Universal Robots URScript: azat-test-new.script

def azattestnew():
  set_gravity([0.0, 0.0, 9.82])
  set_safety_mode_transition_hardness(1)
  set_target_payload(1.070000, [0.002000, 0.003000, 0.057000], [0.001723, 0.001723, 0.001723, 0.000000, 0.000000, 0.000000])
  step_count_12e684db_e6cc_44c8_bfb7_09d4b2be2b77 = 0.0
  thread Step_Counter_Thread_decf62d9_1c1e_413a_991a_3884a730e61c():
    while (True):
      step_count_12e684db_e6cc_44c8_bfb7_09d4b2be2b77 = step_count_12e684db_e6cc_44c8_bfb7_09d4b2be2b77 + 1.0
      sync()
    end
  end
  run Step_Counter_Thread_decf62d9_1c1e_413a_991a_3884a730e61c()
  set_tool_communication(True, 1000000, 2, 1, 1.5, 3.5)
  set_tool_output_mode(0)
  set_tool_digital_output_mode(0, 1)
  set_tool_digital_output_mode(1, 1)
  set_tool_voltage(0)
  set_standard_analog_input_domain(0, 1)
  set_standard_analog_input_domain(1, 1)
  set_tool_analog_input_domain(0, 1)
  set_tool_analog_input_domain(1, 1)
  set_analog_outputdomain(0, 0)
  set_analog_outputdomain(1, 0)
  set_input_actions_to_default()
  set_tcp(p[0.0,0.0,0.0,0.0,0.0,0.0])
  global Plane_1=p[-0.700006141123905,1.3454883874109249E-6,0.3910559577028425,-1.2089868272251132,-1.2089999932245832,1.20858562628424]
  global Plane_2=p[0.0,0.0,0.0,0.0,0.0,0.0]
  global Point_1=p[0.6913645118948067,-0.12399382748223003,0.49223711947071,-1.2983729986843258,1.1259514972191385,-1.2203503861141718]
  $ 1 "Robot Program"
  $ 2 "Script: bookmark_jonathan.script"
  def Machining1():
    # Default parameters:
    global speed_ms = 0.3
    global speed_rads = 0.75
    global accel_mss = 3
    global accel_radss = 1.2
    global blend_radius_m = 0.001

    # Add subprograms here
    # Start of main program
    # Program generated by RoboDK v5.6.5 for UR10e on 13/10/2023 15:41:24
    # Using nominal kinematics.
    blend_radius_m = 0.001
    speed_ms = 1.000
    # set_reference(p[0.335000, -0.154000, 0.001500, 0.000000, 0.000000, 0.000000])
    set_tcp(p[0.000000, 0.000000, 0.252000, 0.000000, 0.000000, 0.000000])
    # Show Tool
    movej([0.110042, -1.089243, -2.581851, -1.041295, 1.570796, 1.680839],accel_radss,speed_rads,0,blend_radius_m)
    movel([0.110042, -1.182009, -2.646989, -0.883391, 1.570796, 1.680839],accel_mss,speed_ms,0,blend_radius_m)
    speed_ms = 1.000
    movel([0.110042, -1.209222, -2.661511, -0.841656, 1.570796, 1.680839],accel_mss,speed_ms,0,blend_radius_m)
    speed_ms = 0.003
    movel([0.110042, -1.219969, -2.666830, -0.825590, 1.570796, 1.680839],accel_mss,speed_ms,0,blend_radius_m)
    speed_ms = 0.007
    movel([0.109778, -1.220368, -2.666631, -0.825390, 1.570796, 1.680574],accel_mss,speed_ms,0,blend_radius_m)
    movel([0.108896, -1.220713, -2.666459, -0.825217, 1.570796, 1.679693],accel_mss,speed_ms,0,blend_radius_m)
    movel([0.108041, -1.221013, -2.666309, -0.825067, 1.570796, 1.678837],accel_mss,speed_ms,0,blend_radius_m)
    movel([0.107066, -1.221345, -2.666143, -0.824901, 1.570796, 1.677863],accel_mss,speed_ms,0,blend_radius_m)
    movel([0.105797, -1.221762, -2.665934, -0.824693, 1.570796, 1.676593],accel_mss,speed_ms,0,blend_radius_m)
    movel([0.105050, -1.221982, -2.665824, -0.824583, 1.570796, 1.675846],accel_mss,speed_ms,0,blend_radius_m)
    movel([0.104582, -1.222084, -2.665773, -0.824532, 1.570796, 1.675378],accel_mss,speed_ms,0,blend_radius_m)
    movel([0.104339, -1.221931, -2.665850, -0.824608, 1.570796, 1.675136],accel_mss,speed_ms,0,blend_radius_m)
    movel([0.104313, -1.221582, -2.666024, -0.824782, 1.570796, 1.675109],accel_mss,speed_ms,0,blend_radius_m)
    movel([0.104310, -1.221133, -2.666249, -0.825007, 1.570796, 1.675106],accel_mss,speed_ms,0,blend_radius_m)
    movel([0.104335, -1.220607, -2.666512, -0.825270, 1.570796, 1.675132],accel_mss,speed_ms,0,blend_radius_m)
    movel([0.104393, -1.219927, -2.666851, -0.825611, 1.570796, 1.675190],accel_mss,speed_ms,0,blend_radius_m)
    movel([0.104458, -1.219512, -2.667058, -0.825819, 1.570796, 1.675255],accel_mss,speed_ms,0,blend_radius_m)
    movel([0.104671, -1.219046, -2.667290, -0.826053, 1.570796, 1.675468],accel_mss,speed_ms,0,blend_radius_m)
    movel([0.104983, -1.218876, -2.667375, -0.826139, 1.570796, 1.675780],accel_mss,speed_ms,0,blend_radius_m)
    movel([0.105336, -1.218982, -2.667322, -0.826085, 1.570796, 1.676132],accel_mss,speed_ms,0,blend_radius_m)
    movel([0.105719, -1.218905, -2.667360, -0.826124, 1.570796, 1.676515],accel_mss,speed_ms,0,blend_radius_m)
    movel([0.106129, -1.218813, -2.667406, -0.826170, 1.570796, 1.676925],accel_mss,speed_ms,0,blend_radius_m)
    movel([0.106457, -1.218831, -2.667397, -0.826161, 1.570796, 1.677253],accel_mss,speed_ms,0,blend_radius_m)
    movel([0.106802, -1.218829, -2.667398, -0.826162, 1.570796, 1.677598],accel_mss,speed_ms,0,blend_radius_m)
    movel([0.107299, -1.218637, -2.667493, -0.826259, 1.570796, 1.678095],accel_mss,speed_ms,0,blend_radius_m)
    movel([0.107817, -1.218437, -2.667593, -0.826359, 1.570796, 1.678614],accel_mss,speed_ms,0,blend_radius_m)
    movel([0.108199, -1.218441, -2.667591, -0.826357, 1.570796, 1.678995],accel_mss,speed_ms,0,blend_radius_m)
    movel([0.108539, -1.218479, -2.667572, -0.826338, 1.570796, 1.679335],accel_mss,speed_ms,0,blend_radius_m)
    movel([0.108879, -1.218392, -2.667615, -0.826382, 1.570796, 1.679675],accel_mss,speed_ms,0,blend_radius_m)
    movel([0.109256, -1.218165, -2.667728, -0.826496, 1.570796, 1.680053],accel_mss,speed_ms,0,blend_radius_m)
    movel([0.109705, -1.217777, -2.667921, -0.826692, 1.570796, 1.680502],accel_mss,speed_ms,0,blend_radius_m)
    movel([0.110106, -1.217433, -2.668091, -0.826865, 1.570796, 1.680902],accel_mss,speed_ms,0,blend_radius_m)
    movel([0.110486, -1.217183, -2.668215, -0.826991, 1.570796, 1.681283],accel_mss,speed_ms,0,blend_radius_m)
    movel([0.110803, -1.217055, -2.668278, -0.827056, 1.570796, 1.681599],accel_mss,speed_ms,0,blend_radius_m)
    movel([0.111053, -1.217213, -2.668200, -0.826976, 1.570796, 1.681849],accel_mss,speed_ms,0,blend_radius_m)
    movel([0.110944, -1.217659, -2.667979, -0.826751, 1.570796, 1.681740],accel_mss,speed_ms,0,blend_radius_m)
    movel([0.110733, -1.218302, -2.667660, -0.826427, 1.570796, 1.681529],accel_mss,speed_ms,0,blend_radius_m)
    movel([0.110389, -1.219201, -2.667213, -0.825975, 1.570796, 1.681186],accel_mss,speed_ms,0,blend_radius_m)
    movel([0.110219, -1.219606, -2.667011, -0.825772, 1.570796, 1.681015],accel_mss,speed_ms,0,blend_radius_m)
    movel([0.110042, -1.219969, -2.666830, -0.825590, 1.570796, 1.680839],accel_mss,speed_ms,0,blend_radius_m)
    speed_ms = 0.003
    movel([0.110042, -1.223618, -2.668588, -0.820184, 1.570796, 1.680839],accel_mss,speed_ms,0,blend_radius_m)
    speed_ms = 0.007
    movel([0.109778, -1.224016, -2.668388, -0.819985, 1.570796, 1.680574],accel_mss,speed_ms,0,blend_radius_m)
    movel([0.108896, -1.224361, -2.668215, -0.819813, 1.570796, 1.679693],accel_mss,speed_ms,0,blend_radius_m)
    movel([0.108041, -1.224660, -2.668065, -0.819664, 1.570796, 1.678837],accel_mss,speed_ms,0,blend_radius_m)
    movel([0.107066, -1.224992, -2.667898, -0.819499, 1.570796, 1.677863],accel_mss,speed_ms,0,blend_radius_m)
    movel([0.105797, -1.225409, -2.667688, -0.819292, 1.570796, 1.676593],accel_mss,speed_ms,0,blend_radius_m)
    movel([0.105050, -1.225628, -2.667578, -0.819183, 1.570796, 1.675846],accel_mss,speed_ms,0,blend_radius_m)
    movel([0.104582, -1.225730, -2.667526, -0.819132, 1.570796, 1.675378],accel_mss,speed_ms,0,blend_radius_m)
    movel([0.104339, -1.225577, -2.667604, -0.819209, 1.570796, 1.675136],accel_mss,speed_ms,0,blend_radius_m)
    movel([0.104313, -1.225229, -2.667779, -0.819381, 1.570796, 1.675109],accel_mss,speed_ms,0,blend_radius_m)
    movel([0.104310, -1.224781, -2.668004, -0.819604, 1.570796, 1.675106],accel_mss,speed_ms,0,blend_radius_m)
    movel([0.104335, -1.224255, -2.668268, -0.819866, 1.570796, 1.675132],accel_mss,speed_ms,0,blend_radius_m)
    movel([0.104393, -1.223576, -2.668608, -0.820205, 1.570796, 1.675190],accel_mss,speed_ms,0,blend_radius_m)
    movel([0.104458, -1.223162, -2.668816, -0.820411, 1.570796, 1.675255],accel_mss,speed_ms,0,blend_radius_m)
    movel([0.104671, -1.222696, -2.669049, -0.820644, 1.570796, 1.675468],accel_mss,speed_ms,0,blend_radius_m)
    movel([0.104983, -1.222527, -2.669134, -0.820729, 1.570796, 1.675780],accel_mss,speed_ms,0,blend_radius_m)
    movel([0.105336, -1.222632, -2.669081, -0.820676, 1.570796, 1.676132],accel_mss,speed_ms,0,blend_radius_m)
    movel([0.105719, -1.222556, -2.669119, -0.820714, 1.570796, 1.676515],accel_mss,speed_ms,0,blend_radius_m)
    movel([0.106129, -1.222464, -2.669165, -0.820760, 1.570796, 1.676925],accel_mss,speed_ms,0,blend_radius_m)
    movel([0.106457, -1.222482, -2.669156, -0.820751, 1.570796, 1.677253],accel_mss,speed_ms,0,blend_radius_m)
    movel([0.106802, -1.222480, -2.669157, -0.820752, 1.570796, 1.677598],accel_mss,speed_ms,0,blend_radius_m)
    movel([0.107299, -1.222288, -2.669253, -0.820848, 1.570796, 1.678095],accel_mss,speed_ms,0,blend_radius_m)
    movel([0.107817, -1.222089, -2.669352, -0.820948, 1.570796, 1.678614],accel_mss,speed_ms,0,blend_radius_m)
    movel([0.108199, -1.222093, -2.669350, -0.820946, 1.570796, 1.678995],accel_mss,speed_ms,0,blend_radius_m)
    movel([0.108539, -1.222130, -2.669332, -0.820927, 1.570796, 1.679335],accel_mss,speed_ms,0,blend_radius_m)
    movel([0.108879, -1.222044, -2.669375, -0.820970, 1.570796, 1.679675],accel_mss,speed_ms,0,blend_radius_m)
    movel([0.109256, -1.221817, -2.669488, -0.821084, 1.570796, 1.680053],accel_mss,speed_ms,0,blend_radius_m)
    movel([0.109705, -1.221429, -2.669681, -0.821278, 1.570796, 1.680502],accel_mss,speed_ms,0,blend_radius_m)
    movel([0.110106, -1.221086, -2.669853, -0.821451, 1.570796, 1.680902],accel_mss,speed_ms,0,blend_radius_m)
    movel([0.110486, -1.220837, -2.669977, -0.821576, 1.570796, 1.681283],accel_mss,speed_ms,0,blend_radius_m)
    movel([0.110803, -1.220709, -2.670040, -0.821640, 1.570796, 1.681599],accel_mss,speed_ms,0,blend_radius_m)
    movel([0.111053, -1.220867, -2.669962, -0.821560, 1.570796, 1.681849],accel_mss,speed_ms,0,blend_radius_m)
    movel([0.110944, -1.221311, -2.669740, -0.821337, 1.570796, 1.681740],accel_mss,speed_ms,0,blend_radius_m)
    movel([0.110733, -1.221954, -2.669420, -0.821016, 1.570796, 1.681529],accel_mss,speed_ms,0,blend_radius_m)
    movel([0.110389, -1.222851, -2.668971, -0.820566, 1.570796, 1.681186],accel_mss,speed_ms,0,blend_radius_m)
    movel([0.110219, -1.223256, -2.668769, -0.820364, 1.570796, 1.681015],accel_mss,speed_ms,0,blend_radius_m)
    movel([0.110042, -1.223618, -2.668588, -0.820184, 1.570796, 1.680839],accel_mss,speed_ms,0,blend_radius_m)
    speed_ms = 0.003
    movel([0.110042, -1.209222, -2.661511, -0.841656, 1.570796, 1.680839],accel_mss,speed_ms,0,blend_radius_m)
    speed_ms = 1.000
    movel([0.110042, -1.182009, -2.646989, -0.883391, 1.570796, 1.680839],accel_mss,speed_ms,0,blend_radius_m)
    movel([0.111003, -1.181848, -2.647065, -0.883476, 1.570796, 1.681799],accel_mss,speed_ms,0,blend_radius_m)
    movel([0.111003, -1.209062, -2.661590, -0.841737, 1.570796, 1.681799],accel_mss,speed_ms,0,blend_radius_m)
    speed_ms = 0.003
    movel([0.111003, -1.219809, -2.666910, -0.825670, 1.570796, 1.681799],accel_mss,speed_ms,0,blend_radius_m)
    speed_ms = 0.007
    movel([0.111091, -1.219320, -2.667153, -0.825915, 1.570796, 1.681888],accel_mss,speed_ms,0,blend_radius_m)
    movel([0.111656, -1.217631, -2.667993, -0.826765, 1.570796, 1.682452],accel_mss,speed_ms,0,blend_radius_m)
    movel([0.112294, -1.215566, -2.669014, -0.827808, 1.570796, 1.683091],accel_mss,speed_ms,0,blend_radius_m)
    movel([0.112472, -1.214337, -2.669620, -0.828432, 1.570796, 1.683268],accel_mss,speed_ms,0,blend_radius_m)
    movel([0.112175, -1.214317, -2.669630, -0.828442, 1.570796, 1.682972],accel_mss,speed_ms,0,blend_radius_m)
    movel([0.111647, -1.214982, -2.669302, -0.828104, 1.570796, 1.682443],accel_mss,speed_ms,0,blend_radius_m)
    movel([0.111241, -1.215691, -2.668953, -0.827745, 1.570796, 1.682038],accel_mss,speed_ms,0,blend_radius_m)
    movel([0.110846, -1.215840, -2.668879, -0.827670, 1.570796, 1.681643],accel_mss,speed_ms,0,blend_radius_m)
    movel([0.110875, -1.215298, -2.669147, -0.827944, 1.570796, 1.681671],accel_mss,speed_ms,0,blend_radius_m)
    movel([0.110894, -1.214637, -2.669473, -0.828280, 1.570796, 1.681690],accel_mss,speed_ms,0,blend_radius_m)
    movel([0.110778, -1.214112, -2.669731, -0.828546, 1.570796, 1.681574],accel_mss,speed_ms,0,blend_radius_m)
    movel([0.110562, -1.213807, -2.669881, -0.828701, 1.570796, 1.681358],accel_mss,speed_ms,0,blend_radius_m)
    movel([0.110274, -1.213811, -2.669879, -0.828699, 1.570796, 1.681070],accel_mss,speed_ms,0,blend_radius_m)
    movel([0.109960, -1.214075, -2.669749, -0.828565, 1.570796, 1.680756],accel_mss,speed_ms,0,blend_radius_m)
    movel([0.109672, -1.214507, -2.669536, -0.828345, 1.570796, 1.680469],accel_mss,speed_ms,0,blend_radius_m)
    movel([0.109450, -1.214884, -2.669351, -0.828154, 1.570796, 1.680246],accel_mss,speed_ms,0,blend_radius_m)
    movel([0.109129, -1.214990, -2.669298, -0.828100, 1.570796, 1.679926],accel_mss,speed_ms,0,blend_radius_m)
    movel([0.109040, -1.214717, -2.669433, -0.828239, 1.570796, 1.679836],accel_mss,speed_ms,0,blend_radius_m)
    movel([0.108872, -1.214255, -2.669661, -0.828473, 1.570796, 1.679668],accel_mss,speed_ms,0,blend_radius_m)
    movel([0.108592, -1.214163, -2.669706, -0.828520, 1.570796, 1.679388],accel_mss,speed_ms,0,blend_radius_m)
    movel([0.108228, -1.214389, -2.669594, -0.828405, 1.570796, 1.679024],accel_mss,speed_ms,0,blend_radius_m)
    movel([0.107783, -1.214975, -2.669306, -0.828108, 1.570796, 1.678580],accel_mss,speed_ms,0,blend_radius_m)
    movel([0.107321, -1.215692, -2.668952, -0.827745, 1.570796, 1.678117],accel_mss,speed_ms,0,blend_radius_m)
    movel([0.106937, -1.215475, -2.669060, -0.827855, 1.570796, 1.677734],accel_mss,speed_ms,0,blend_radius_m)
    movel([0.106603, -1.215377, -2.669108, -0.827904, 1.570796, 1.677399],accel_mss,speed_ms,0,blend_radius_m)
    movel([0.106283, -1.215476, -2.669059, -0.827854, 1.570796, 1.677080],accel_mss,speed_ms,0,blend_radius_m)
    movel([0.105977, -1.215764, -2.668917, -0.827708, 1.570796, 1.676773],accel_mss,speed_ms,0,blend_radius_m)
    movel([0.105684, -1.216259, -2.668672, -0.827458, 1.570796, 1.676480],accel_mss,speed_ms,0,blend_radius_m)
    movel([0.105478, -1.216605, -2.668501, -0.827283, 1.570796, 1.676274],accel_mss,speed_ms,0,blend_radius_m)
    movel([0.105093, -1.216818, -2.668396, -0.827175, 1.570796, 1.675890],accel_mss,speed_ms,0,blend_radius_m)
    movel([0.104873, -1.216441, -2.668582, -0.827366, 1.570796, 1.675669],accel_mss,speed_ms,0,blend_radius_m)
    movel([0.104483, -1.216372, -2.668616, -0.827401, 1.570796, 1.675279],accel_mss,speed_ms,0,blend_radius_m)
    movel([0.104111, -1.216774, -2.668417, -0.827197, 1.570796, 1.674908],accel_mss,speed_ms,0,blend_radius_m)
    movel([0.103999, -1.217250, -2.668181, -0.826957, 1.570796, 1.674795],accel_mss,speed_ms,0,blend_radius_m)
    movel([0.103883, -1.218034, -2.667793, -0.826562, 1.570796, 1.674679],accel_mss,speed_ms,0,blend_radius_m)
    movel([0.103712, -1.219580, -2.667024, -0.825785, 1.570796, 1.674509],accel_mss,speed_ms,0,blend_radius_m)
    movel([0.103592, -1.220658, -2.666486, -0.825245, 1.570796, 1.674388],accel_mss,speed_ms,0,blend_radius_m)
    movel([0.103471, -1.221596, -2.666018, -0.824776, 1.570796, 1.674267],accel_mss,speed_ms,0,blend_radius_m)
    movel([0.103356, -1.222403, -2.665613, -0.824373, 1.570796, 1.674152],accel_mss,speed_ms,0,blend_radius_m)
    movel([0.103121, -1.222715, -2.665456, -0.824217, 1.570796, 1.673917],accel_mss,speed_ms,0,blend_radius_m)
    movel([0.102527, -1.222915, -2.665357, -0.824118, 1.570796, 1.673323],accel_mss,speed_ms,0,blend_radius_m)
    movel([0.102201, -1.222577, -2.665526, -0.824286, 1.570796, 1.672997],accel_mss,speed_ms,0,blend_radius_m)
    movel([0.102154, -1.221734, -2.665948, -0.824707, 1.570796, 1.672951],accel_mss,speed_ms,0,blend_radius_m)
    movel([0.102170, -1.220698, -2.666466, -0.825224, 1.570796, 1.672966],accel_mss,speed_ms,0,blend_radius_m)
    movel([0.102265, -1.219574, -2.667027, -0.825788, 1.570796, 1.673061],accel_mss,speed_ms,0,blend_radius_m)
    movel([0.102925, -1.216505, -2.668551, -0.827334, 1.570796, 1.673721],accel_mss,speed_ms,0,blend_radius_m)
    movel([0.104167, -1.213999, -2.669786, -0.828603, 1.570796, 1.674963],accel_mss,speed_ms,0,blend_radius_m)
    movel([0.106022, -1.212020, -2.670758, -0.829611, 1.570796, 1.676818],accel_mss,speed_ms,0,blend_radius_m)
    movel([0.108479, -1.210505, -2.671498, -0.830386, 1.570796, 1.679276],accel_mss,speed_ms,0,blend_radius_m)
    movel([0.109965, -1.209971, -2.671759, -0.830659, 1.570796, 1.680761],accel_mss,speed_ms,0,blend_radius_m)
    movel([0.111428, -1.209723, -2.671880, -0.830787, 1.570796, 1.682224],accel_mss,speed_ms,0,blend_radius_m)
    movel([0.112682, -1.209773, -2.671855, -0.830761, 1.570796, 1.683478],accel_mss,speed_ms,0,blend_radius_m)
    movel([0.113540, -1.210140, -2.671676, -0.830573, 1.570796, 1.684337],accel_mss,speed_ms,0,blend_radius_m)
    movel([0.114168, -1.210944, -2.671284, -0.830161, 1.570796, 1.684965],accel_mss,speed_ms,0,blend_radius_m)
    movel([0.114448, -1.212086, -2.670725, -0.829577, 1.570796, 1.685244],accel_mss,speed_ms,0,blend_radius_m)
    movel([0.114379, -1.213608, -2.669979, -0.828802, 1.570796, 1.685175],accel_mss,speed_ms,0,blend_radius_m)
    movel([0.113959, -1.215557, -2.669019, -0.827813, 1.570796, 1.684755],accel_mss,speed_ms,0,blend_radius_m)
    movel([0.113608, -1.216725, -2.668442, -0.827222, 1.570796, 1.684404],accel_mss,speed_ms,0,blend_radius_m)
    movel([0.113186, -1.217929, -2.667845, -0.826615, 1.570796, 1.683983],accel_mss,speed_ms,0,blend_radius_m)
    movel([0.112766, -1.218994, -2.667316, -0.826079, 1.570796, 1.683562],accel_mss,speed_ms,0,blend_radius_m)
    movel([0.112498, -1.219453, -2.667088, -0.825849, 1.570796, 1.683295],accel_mss,speed_ms,0,blend_radius_m)
    movel([0.112181, -1.219683, -2.666973, -0.825733, 1.570796, 1.682978],accel_mss,speed_ms,0,blend_radius_m)
    movel([0.111627, -1.219898, -2.666865, -0.825625, 1.570796, 1.682423],accel_mss,speed_ms,0,blend_radius_m)
    movel([0.111159, -1.219969, -2.666830, -0.825590, 1.570796, 1.681956],accel_mss,speed_ms,0,blend_radius_m)
    movel([0.111003, -1.219809, -2.666910, -0.825670, 1.570796, 1.681799],accel_mss,speed_ms,0,blend_radius_m)
    speed_ms = 0.003
    movel([0.111003, -1.223459, -2.668667, -0.820263, 1.570796, 1.681799],accel_mss,speed_ms,0,blend_radius_m)
    speed_ms = 0.007
    movel([0.111091, -1.222970, -2.668912, -0.820507, 1.570796, 1.681888],accel_mss,speed_ms,0,blend_radius_m)
    movel([0.111656, -1.221284, -2.669754, -0.821351, 1.570796, 1.682452],accel_mss,speed_ms,0,blend_radius_m)
    movel([0.112294, -1.219222, -2.670779, -0.822388, 1.570796, 1.683091],accel_mss,speed_ms,0,blend_radius_m)
    movel([0.112472, -1.217995, -2.671387, -0.823007, 1.570796, 1.683268],accel_mss,speed_ms,0,blend_radius_m)
    movel([0.112175, -1.217975, -2.671397, -0.823017, 1.570796, 1.682972],accel_mss,speed_ms,0,blend_radius_m)
    movel([0.111647, -1.218639, -2.671068, -0.822681, 1.570796, 1.682443],accel_mss,speed_ms,0,blend_radius_m)
    movel([0.111241, -1.219347, -2.670717, -0.822325, 1.570796, 1.682038],accel_mss,speed_ms,0,blend_radius_m)
    movel([0.110846, -1.219495, -2.670644, -0.822250, 1.570796, 1.681643],accel_mss,speed_ms,0,blend_radius_m)
    movel([0.110875, -1.218954, -2.670912, -0.822523, 1.570796, 1.681671],accel_mss,speed_ms,0,blend_radius_m)
    movel([0.110894, -1.218294, -2.671239, -0.822856, 1.570796, 1.681690],accel_mss,speed_ms,0,blend_radius_m)
    movel([0.110778, -1.217770, -2.671498, -0.823120, 1.570796, 1.681574],accel_mss,speed_ms,0,blend_radius_m)
    movel([0.110562, -1.217466, -2.671649, -0.823274, 1.570796, 1.681358],accel_mss,speed_ms,0,blend_radius_m)
    movel([0.110274, -1.217470, -2.671647, -0.823272, 1.570796, 1.681070],accel_mss,speed_ms,0,blend_radius_m)
    movel([0.109960, -1.217733, -2.671517, -0.823139, 1.570796, 1.680756],accel_mss,speed_ms,0,blend_radius_m)
    movel([0.109672, -1.218165, -2.671303, -0.822921, 1.570796, 1.680469],accel_mss,speed_ms,0,blend_radius_m)
    movel([0.109450, -1.218541, -2.671117, -0.822731, 1.570796, 1.680246],accel_mss,speed_ms,0,blend_radius_m)
    movel([0.109129, -1.218647, -2.671064, -0.822678, 1.570796, 1.679926],accel_mss,speed_ms,0,blend_radius_m)
    movel([0.109040, -1.218375, -2.671199, -0.822815, 1.570796, 1.679836],accel_mss,speed_ms,0,blend_radius_m)
    movel([0.108872, -1.217913, -2.671428, -0.823048, 1.570796, 1.679668],accel_mss,speed_ms,0,blend_radius_m)
    movel([0.108592, -1.217821, -2.671473, -0.823095, 1.570796, 1.679388],accel_mss,speed_ms,0,blend_radius_m)
    movel([0.108228, -1.218047, -2.671361, -0.822980, 1.570796, 1.679024],accel_mss,speed_ms,0,blend_radius_m)
    movel([0.107783, -1.218632, -2.671072, -0.822685, 1.570796, 1.678580],accel_mss,speed_ms,0,blend_radius_m)
    movel([0.107321, -1.219348, -2.670717, -0.822324, 1.570796, 1.678117],accel_mss,speed_ms,0,blend_radius_m)
    movel([0.106937, -1.219131, -2.670824, -0.822434, 1.570796, 1.677734],accel_mss,speed_ms,0,blend_radius_m)
    movel([0.106603, -1.219033, -2.670873, -0.822483, 1.570796, 1.677399],accel_mss,speed_ms,0,blend_radius_m)
    movel([0.106283, -1.219132, -2.670824, -0.822433, 1.570796, 1.677080],accel_mss,speed_ms,0,blend_radius_m)
    movel([0.105977, -1.219420, -2.670681, -0.822288, 1.570796, 1.676773],accel_mss,speed_ms,0,blend_radius_m)
    movel([0.105684, -1.219914, -2.670436, -0.822039, 1.570796, 1.676480],accel_mss,speed_ms,0,blend_radius_m)
    movel([0.105478, -1.220260, -2.670264, -0.821865, 1.570796, 1.676274],accel_mss,speed_ms,0,blend_radius_m)
    movel([0.105093, -1.220472, -2.670158, -0.821759, 1.570796, 1.675890],accel_mss,speed_ms,0,blend_radius_m)
    movel([0.104873, -1.220095, -2.670345, -0.821948, 1.570796, 1.675669],accel_mss,speed_ms,0,blend_radius_m)
    movel([0.104483, -1.220027, -2.670379, -0.821982, 1.570796, 1.675279],accel_mss,speed_ms,0,blend_radius_m)
    movel([0.104111, -1.220429, -2.670180, -0.821781, 1.570796, 1.674908],accel_mss,speed_ms,0,blend_radius_m)
    movel([0.103999, -1.220904, -2.669943, -0.821542, 1.570796, 1.674795],accel_mss,speed_ms,0,blend_radius_m)
    movel([0.103883, -1.221687, -2.669553, -0.821149, 1.570796, 1.674679],accel_mss,speed_ms,0,blend_radius_m)
    movel([0.103712, -1.223230, -2.668782, -0.820377, 1.570796, 1.674509],accel_mss,speed_ms,0,blend_radius_m)
    movel([0.103592, -1.224306, -2.668242, -0.819840, 1.570796, 1.674388],accel_mss,speed_ms,0,blend_radius_m)
    movel([0.103471, -1.225242, -2.667772, -0.819375, 1.570796, 1.674267],accel_mss,speed_ms,0,blend_radius_m)
    movel([0.103356, -1.226049, -2.667366, -0.818974, 1.570796, 1.674152],accel_mss,speed_ms,0,blend_radius_m)
    movel([0.103121, -1.226360, -2.667209, -0.818820, 1.570796, 1.673917],accel_mss,speed_ms,0,blend_radius_m)
    movel([0.102527, -1.226559, -2.667109, -0.818721, 1.570796, 1.673323],accel_mss,speed_ms,0,blend_radius_m)
    movel([0.102201, -1.226222, -2.667279, -0.818889, 1.570796, 1.672997],accel_mss,speed_ms,0,blend_radius_m)
    movel([0.102154, -1.225380, -2.667703, -0.819306, 1.570796, 1.672951],accel_mss,speed_ms,0,blend_radius_m)
    movel([0.102170, -1.224346, -2.668222, -0.819820, 1.570796, 1.672966],accel_mss,speed_ms,0,blend_radius_m)
    movel([0.102265, -1.223224, -2.668785, -0.820380, 1.570796, 1.673061],accel_mss,speed_ms,0,blend_radius_m)
    movel([0.102925, -1.220160, -2.670314, -0.821916, 1.570796, 1.673721],accel_mss,speed_ms,0,blend_radius_m)
    movel([0.104167, -1.217658, -2.671554, -0.823177, 1.570796, 1.674963],accel_mss,speed_ms,0,blend_radius_m)
    movel([0.106022, -1.215681, -2.672529, -0.824179, 1.570796, 1.676818],accel_mss,speed_ms,0,blend_radius_m)
    movel([0.108479, -1.214169, -2.673272, -0.824949, 1.570796, 1.679276],accel_mss,speed_ms,0,blend_radius_m)
    movel([0.109965, -1.213636, -2.673533, -0.825220, 1.570796, 1.680761],accel_mss,speed_ms,0,blend_radius_m)
    movel([0.111428, -1.213388, -2.673654, -0.825347, 1.570796, 1.682224],accel_mss,speed_ms,0,blend_radius_m)
    movel([0.112682, -1.213438, -2.673630, -0.825322, 1.570796, 1.683478],accel_mss,speed_ms,0,blend_radius_m)
    movel([0.113540, -1.213804, -2.673450, -0.825135, 1.570796, 1.684337],accel_mss,speed_ms,0,blend_radius_m)
    movel([0.114168, -1.214608, -2.673056, -0.824725, 1.570796, 1.684965],accel_mss,speed_ms,0,blend_radius_m)
    movel([0.114448, -1.215748, -2.672496, -0.824145, 1.570796, 1.685244],accel_mss,speed_ms,0,blend_radius_m)
    movel([0.114379, -1.217268, -2.671747, -0.823375, 1.570796, 1.685175],accel_mss,speed_ms,0,blend_radius_m)
    movel([0.113959, -1.219213, -2.670784, -0.822392, 1.570796, 1.684755],accel_mss,speed_ms,0,blend_radius_m)
    movel([0.113608, -1.220379, -2.670204, -0.821805, 1.570796, 1.684404],accel_mss,speed_ms,0,blend_radius_m)
    movel([0.113186, -1.221582, -2.669605, -0.821202, 1.570796, 1.683983],accel_mss,speed_ms,0,blend_radius_m)
    movel([0.112766, -1.222645, -2.669074, -0.820670, 1.570796, 1.683562],accel_mss,speed_ms,0,blend_radius_m)
    movel([0.112498, -1.223103, -2.668846, -0.820441, 1.570796, 1.683295],accel_mss,speed_ms,0,blend_radius_m)
    movel([0.112181, -1.223333, -2.668730, -0.820326, 1.570796, 1.682978],accel_mss,speed_ms,0,blend_radius_m)
    movel([0.111627, -1.223548, -2.668623, -0.820219, 1.570796, 1.682423],accel_mss,speed_ms,0,blend_radius_m)
    movel([0.111159, -1.223618, -2.668587, -0.820183, 1.570796, 1.681956],accel_mss,speed_ms,0,blend_radius_m)
    movel([0.111003, -1.223459, -2.668667, -0.820263, 1.570796, 1.681799],accel_mss,speed_ms,0,blend_radius_m)
    speed_ms = 0.003
    movel([0.111003, -1.209062, -2.661590, -0.841737, 1.570796, 1.681799],accel_mss,speed_ms,0,blend_radius_m)
    speed_ms = 1.000
    movel([0.111003, -1.181848, -2.647065, -0.883476, 1.570796, 1.681799],accel_mss,speed_ms,0,blend_radius_m)
    movel([0.109065, -1.179479, -2.648185, -0.884725, 1.570796, 1.679861],accel_mss,speed_ms,0,blend_radius_m)
    movel([0.109065, -1.206712, -2.662741, -0.842936, 1.570796, 1.679861],accel_mss,speed_ms,0,blend_radius_m)
    speed_ms = 0.003
    movel([0.109065, -1.217469, -2.668073, -0.826847, 1.570796, 1.679861],accel_mss,speed_ms,0,blend_radius_m)
    speed_ms = 0.007
    movel([0.108578, -1.217519, -2.668048, -0.826821, 1.570796, 1.679374],accel_mss,speed_ms,0,blend_radius_m)
    movel([0.108509, -1.217274, -2.668170, -0.826945, 1.570796, 1.679305],accel_mss,speed_ms,0,blend_radius_m)
    movel([0.108593, -1.216907, -2.668352, -0.827130, 1.570796, 1.679389],accel_mss,speed_ms,0,blend_radius_m)
    movel([0.108773, -1.216518, -2.668544, -0.827327, 1.570796, 1.679569],accel_mss,speed_ms,0,blend_radius_m)
    movel([0.109113, -1.216290, -2.668657, -0.827442, 1.570796, 1.679909],accel_mss,speed_ms,0,blend_radius_m)
    movel([0.109347, -1.216733, -2.668438, -0.827218, 1.570796, 1.680143],accel_mss,speed_ms,0,blend_radius_m)
    movel([0.109341, -1.217024, -2.668294, -0.827071, 1.570796, 1.680137],accel_mss,speed_ms,0,blend_radius_m)
    movel([0.109065, -1.217469, -2.668073, -0.826847, 1.570796, 1.679861],accel_mss,speed_ms,0,blend_radius_m)
    speed_ms = 0.003
    movel([0.109065, -1.221122, -2.669834, -0.821432, 1.570796, 1.679861],accel_mss,speed_ms,0,blend_radius_m)
    speed_ms = 0.007
    movel([0.108578, -1.221172, -2.669809, -0.821407, 1.570796, 1.679374],accel_mss,speed_ms,0,blend_radius_m)
    movel([0.108509, -1.220928, -2.669931, -0.821530, 1.570796, 1.679305],accel_mss,speed_ms,0,blend_radius_m)
    movel([0.108593, -1.220561, -2.670114, -0.821714, 1.570796, 1.679389],accel_mss,speed_ms,0,blend_radius_m)
    movel([0.108773, -1.220172, -2.670307, -0.821909, 1.570796, 1.679569],accel_mss,speed_ms,0,blend_radius_m)
    movel([0.109113, -1.219945, -2.670420, -0.822024, 1.570796, 1.679909],accel_mss,speed_ms,0,blend_radius_m)
    movel([0.109347, -1.220387, -2.670200, -0.821801, 1.570796, 1.680143],accel_mss,speed_ms,0,blend_radius_m)
    movel([0.109341, -1.220678, -2.670056, -0.821655, 1.570796, 1.680137],accel_mss,speed_ms,0,blend_radius_m)
    movel([0.109065, -1.221122, -2.669834, -0.821432, 1.570796, 1.679861],accel_mss,speed_ms,0,blend_radius_m)
    speed_ms = 0.003
    movel([0.109065, -1.206712, -2.662741, -0.842936, 1.570796, 1.679861],accel_mss,speed_ms,0,blend_radius_m)
    speed_ms = 1.000
    movel([0.109065, -1.179479, -2.648185, -0.884725, 1.570796, 1.679861],accel_mss,speed_ms,0,blend_radius_m)
    movel([0.107392, -1.179562, -2.648146, -0.884681, 1.570796, 1.678188],accel_mss,speed_ms,0,blend_radius_m)
    movel([0.107392, -1.206796, -2.662700, -0.842893, 1.570796, 1.678188],accel_mss,speed_ms,0,blend_radius_m)
    speed_ms = 0.003
    movel([0.107392, -1.217552, -2.668032, -0.826805, 1.570796, 1.678188],accel_mss,speed_ms,0,blend_radius_m)
    speed_ms = 0.007
    movel([0.106968, -1.217951, -2.667834, -0.826604, 1.570796, 1.677765],accel_mss,speed_ms,0,blend_radius_m)
    movel([0.106710, -1.217709, -2.667954, -0.826726, 1.570796, 1.677506],accel_mss,speed_ms,0,blend_radius_m)
    movel([0.106767, -1.217397, -2.668109, -0.826883, 1.570796, 1.677563],accel_mss,speed_ms,0,blend_radius_m)
    movel([0.107140, -1.217006, -2.668303, -0.827081, 1.570796, 1.677937],accel_mss,speed_ms,0,blend_radius_m)
    movel([0.107318, -1.217145, -2.668234, -0.827011, 1.570796, 1.678115],accel_mss,speed_ms,0,blend_radius_m)
    movel([0.107403, -1.217506, -2.668055, -0.826828, 1.570796, 1.678200],accel_mss,speed_ms,0,blend_radius_m)
    speed_ms = 0.003
    movel([0.107392, -1.221205, -2.669793, -0.821391, 1.570796, 1.678188],accel_mss,speed_ms,0,blend_radius_m)
    speed_ms = 0.007
    movel([0.106968, -1.221603, -2.669595, -0.821191, 1.570796, 1.677765],accel_mss,speed_ms,0,blend_radius_m)
    movel([0.106710, -1.221362, -2.669715, -0.821312, 1.570796, 1.677506],accel_mss,speed_ms,0,blend_radius_m)
    movel([0.106767, -1.221050, -2.669870, -0.821469, 1.570796, 1.677563],accel_mss,speed_ms,0,blend_radius_m)
    movel([0.107140, -1.220659, -2.670065, -0.821665, 1.570796, 1.677937],accel_mss,speed_ms,0,blend_radius_m)
    movel([0.107318, -1.220798, -2.669996, -0.821595, 1.570796, 1.678115],accel_mss,speed_ms,0,blend_radius_m)
    movel([0.107403, -1.221159, -2.669816, -0.821414, 1.570796, 1.678200],accel_mss,speed_ms,0,blend_radius_m)
    speed_ms = 0.003
    movel([0.107392, -1.206796, -2.662700, -0.842893, 1.570796, 1.678188],accel_mss,speed_ms,0,blend_radius_m)
    speed_ms = 1.000
    movel([0.107392, -1.179562, -2.648146, -0.884681, 1.570796, 1.678188],accel_mss,speed_ms,0,blend_radius_m)
    movel([0.090800, -1.186880, -2.644666, -0.880842, 1.570796, 1.661597],accel_mss,speed_ms,0,blend_radius_m)
    movel([0.090800, -1.214052, -2.659125, -0.839212, 1.570796, 1.661597],accel_mss,speed_ms,0,blend_radius_m)
    speed_ms = 0.003
    movel([0.090800, -1.224777, -2.664420, -0.823192, 1.570796, 1.661597],accel_mss,speed_ms,0,blend_radius_m)
    speed_ms = 0.007
    movel([0.090349, -1.225349, -2.664131, -0.822909, 1.570796, 1.661146],accel_mss,speed_ms,0,blend_radius_m)
    movel([0.089579, -1.225816, -2.663895, -0.822678, 1.570796, 1.660376],accel_mss,speed_ms,0,blend_radius_m)
    movel([0.088964, -1.226163, -2.663720, -0.822506, 1.570796, 1.659760],accel_mss,speed_ms,0,blend_radius_m)
    movel([0.087981, -1.226712, -2.663442, -0.822235, 1.570796, 1.658778],accel_mss,speed_ms,0,blend_radius_m)
    movel([0.086862, -1.227338, -2.663125, -0.821926, 1.570796, 1.657659],accel_mss,speed_ms,0,blend_radius_m)
    movel([0.085757, -1.227956, -2.662811, -0.821622, 1.570796, 1.656553],accel_mss,speed_ms,0,blend_radius_m)
    movel([0.084618, -1.228592, -2.662488, -0.821309, 1.570796, 1.655415],accel_mss,speed_ms,0,blend_radius_m)
    movel([0.083401, -1.229276, -2.662140, -0.820973, 1.570796, 1.654198],accel_mss,speed_ms,0,blend_radius_m)
    movel([0.082286, -1.229909, -2.661817, -0.820662, 1.570796, 1.653082],accel_mss,speed_ms,0,blend_radius_m)
    movel([0.081487, -1.230366, -2.661584, -0.820439, 1.570796, 1.652284],accel_mss,speed_ms,0,blend_radius_m)
    movel([0.077430, -1.232696, -2.660391, -0.819301, 1.570796, 1.648226],accel_mss,speed_ms,0,blend_radius_m)
    movel([0.075172, -1.233962, -2.659741, -0.818686, 1.570796, 1.645969],accel_mss,speed_ms,0,blend_radius_m)
    movel([0.073687, -1.234764, -2.659328, -0.818297, 1.570796, 1.644483],accel_mss,speed_ms,0,blend_radius_m)
    movel([0.073372, -1.234811, -2.659304, -0.818275, 1.570796, 1.644168],accel_mss,speed_ms,0,blend_radius_m)
    movel([0.073295, -1.234580, -2.659423, -0.818387, 1.570796, 1.644092],accel_mss,speed_ms,0,blend_radius_m)
    movel([0.073585, -1.234185, -2.659626, -0.818578, 1.570796, 1.644381],accel_mss,speed_ms,0,blend_radius_m)
    movel([0.073559, -1.233831, -2.659808, -0.818750, 1.570796, 1.644355],accel_mss,speed_ms,0,blend_radius_m)
    movel([0.073378, -1.233431, -2.660014, -0.818944, 1.570796, 1.644175],accel_mss,speed_ms,0,blend_radius_m)
    movel([0.073158, -1.232131, -2.660681, -0.819577, 1.570796, 1.643955],accel_mss,speed_ms,0,blend_radius_m)
    movel([0.072974, -1.230711, -2.661408, -0.820270, 1.570796, 1.643770],accel_mss,speed_ms,0,blend_radius_m)
    movel([0.072889, -1.229445, -2.662054, -0.820890, 1.570796, 1.643685],accel_mss,speed_ms,0,blend_radius_m)
    movel([0.072885, -1.228854, -2.662355, -0.821180, 1.570796, 1.643681],accel_mss,speed_ms,0,blend_radius_m)
    movel([0.072909, -1.228198, -2.662689, -0.821503, 1.570796, 1.643705],accel_mss,speed_ms,0,blend_radius_m)
    movel([0.072955, -1.227568, -2.663008, -0.821813, 1.570796, 1.643751],accel_mss,speed_ms,0,blend_radius_m)
    movel([0.073020, -1.227085, -2.663253, -0.822051, 1.570796, 1.643817],accel_mss,speed_ms,0,blend_radius_m)
    movel([0.073121, -1.226456, -2.663571, -0.822361, 1.570796, 1.643917],accel_mss,speed_ms,0,blend_radius_m)
    movel([0.073123, -1.226187, -2.663708, -0.822494, 1.570796, 1.643919],accel_mss,speed_ms,0,blend_radius_m)
    movel([0.072829, -1.225895, -2.663855, -0.822639, 1.570796, 1.643626],accel_mss,speed_ms,0,blend_radius_m)
    movel([0.072567, -1.225713, -2.663948, -0.822729, 1.570796, 1.643364],accel_mss,speed_ms,0,blend_radius_m)
    movel([0.072608, -1.225208, -2.664202, -0.822979, 1.570796, 1.643404],accel_mss,speed_ms,0,blend_radius_m)
    movel([0.072924, -1.224797, -2.664409, -0.823182, 1.570796, 1.643721],accel_mss,speed_ms,0,blend_radius_m)
    movel([0.073226, -1.224392, -2.664614, -0.823383, 1.570796, 1.644022],accel_mss,speed_ms,0,blend_radius_m)
    movel([0.073128, -1.224161, -2.664730, -0.823498, 1.570796, 1.643924],accel_mss,speed_ms,0,blend_radius_m)
    movel([0.073050, -1.223833, -2.664895, -0.823661, 1.570796, 1.643846],accel_mss,speed_ms,0,blend_radius_m)
    movel([0.072942, -1.223512, -2.665057, -0.823821, 1.570796, 1.643738],accel_mss,speed_ms,0,blend_radius_m)
    movel([0.072715, -1.223352, -2.665137, -0.823900, 1.570796, 1.643512],accel_mss,speed_ms,0,blend_radius_m)
    movel([0.072769, -1.222971, -2.665328, -0.824090, 1.570796, 1.643566],accel_mss,speed_ms,0,blend_radius_m)
    movel([0.073235, -1.222419, -2.665605, -0.824365, 1.570796, 1.644032],accel_mss,speed_ms,0,blend_radius_m)
    movel([0.073730, -1.221882, -2.665874, -0.824633, 1.570796, 1.644526],accel_mss,speed_ms,0,blend_radius_m)
    movel([0.074179, -1.221685, -2.665973, -0.824731, 1.570796, 1.644975],accel_mss,speed_ms,0,blend_radius_m)
    movel([0.074415, -1.221763, -2.665934, -0.824692, 1.570796, 1.645212],accel_mss,speed_ms,0,blend_radius_m)
    movel([0.074609, -1.221891, -2.665870, -0.824628, 1.570796, 1.645406],accel_mss,speed_ms,0,blend_radius_m)
    movel([0.074697, -1.222277, -2.665676, -0.824436, 1.570796, 1.645493],accel_mss,speed_ms,0,blend_radius_m)
    movel([0.074870, -1.222553, -2.665538, -0.824298, 1.570796, 1.645666],accel_mss,speed_ms,0,blend_radius_m)
    movel([0.075082, -1.222780, -2.665424, -0.824185, 1.570796, 1.645878],accel_mss,speed_ms,0,blend_radius_m)
    movel([0.075630, -1.222582, -2.665524, -0.824284, 1.570796, 1.646426],accel_mss,speed_ms,0,blend_radius_m)
    movel([0.076550, -1.221927, -2.665852, -0.824611, 1.570796, 1.647346],accel_mss,speed_ms,0,blend_radius_m)
    movel([0.077489, -1.221235, -2.666198, -0.824956, 1.570796, 1.648285],accel_mss,speed_ms,0,blend_radius_m)
    movel([0.077732, -1.220925, -2.666353, -0.825111, 1.570796, 1.648528],accel_mss,speed_ms,0,blend_radius_m)
    movel([0.077653, -1.220659, -2.666486, -0.825244, 1.570796, 1.648449],accel_mss,speed_ms,0,blend_radius_m)
    movel([0.077678, -1.220297, -2.666667, -0.825426, 1.570796, 1.648474],accel_mss,speed_ms,0,blend_radius_m)
    movel([0.077699, -1.220025, -2.666802, -0.825562, 1.570796, 1.648495],accel_mss,speed_ms,0,blend_radius_m)
    movel([0.077413, -1.219642, -2.666993, -0.825754, 1.570796, 1.648209],accel_mss,speed_ms,0,blend_radius_m)
    movel([0.077317, -1.219189, -2.667219, -0.825981, 1.570796, 1.648113],accel_mss,speed_ms,0,blend_radius_m)
    movel([0.077299, -1.218682, -2.667471, -0.826236, 1.570796, 1.648095],accel_mss,speed_ms,0,blend_radius_m)
    movel([0.077389, -1.218280, -2.667671, -0.826438, 1.570796, 1.648186],accel_mss,speed_ms,0,blend_radius_m)
    movel([0.077615, -1.217904, -2.667857, -0.826628, 1.570796, 1.648412],accel_mss,speed_ms,0,blend_radius_m)
    movel([0.078010, -1.217509, -2.668053, -0.826827, 1.570796, 1.648807],accel_mss,speed_ms,0,blend_radius_m)
    movel([0.078613, -1.217060, -2.668276, -0.827053, 1.570796, 1.649409],accel_mss,speed_ms,0,blend_radius_m)
    movel([0.079495, -1.216509, -2.668549, -0.827332, 1.570796, 1.650291],accel_mss,speed_ms,0,blend_radius_m)
    movel([0.080567, -1.215905, -2.668847, -0.827637, 1.570796, 1.651364],accel_mss,speed_ms,0,blend_radius_m)
    movel([0.081345, -1.215546, -2.669024, -0.827818, 1.570796, 1.652142],accel_mss,speed_ms,0,blend_radius_m)
    movel([0.081899, -1.215392, -2.669101, -0.827897, 1.570796, 1.652696],accel_mss,speed_ms,0,blend_radius_m)
    movel([0.082256, -1.215438, -2.669077, -0.827873, 1.570796, 1.653053],accel_mss,speed_ms,0,blend_radius_m)
    movel([0.082498, -1.215684, -2.668956, -0.827749, 1.570796, 1.653294],accel_mss,speed_ms,0,blend_radius_m)
    movel([0.082652, -1.216117, -2.668743, -0.827530, 1.570796, 1.653448],accel_mss,speed_ms,0,blend_radius_m)
    movel([0.082703, -1.216581, -2.668513, -0.827295, 1.570796, 1.653499],accel_mss,speed_ms,0,blend_radius_m)
    movel([0.082589, -1.216924, -2.668343, -0.827122, 1.570796, 1.653386],accel_mss,speed_ms,0,blend_radius_m)
    movel([0.082550, -1.217317, -2.668148, -0.826923, 1.570796, 1.653347],accel_mss,speed_ms,0,blend_radius_m)
    movel([0.082765, -1.217533, -2.668041, -0.826815, 1.570796, 1.653561],accel_mss,speed_ms,0,blend_radius_m)
    movel([0.082850, -1.217759, -2.667929, -0.826701, 1.570796, 1.653646],accel_mss,speed_ms,0,blend_radius_m)
    movel([0.083106, -1.217930, -2.667845, -0.826615, 1.570796, 1.653902],accel_mss,speed_ms,0,blend_radius_m)
    movel([0.083419, -1.217835, -2.667892, -0.826662, 1.570796, 1.654215],accel_mss,speed_ms,0,blend_radius_m)
    movel([0.083853, -1.217665, -2.667976, -0.826748, 1.570796, 1.654650],accel_mss,speed_ms,0,blend_radius_m)
    movel([0.084433, -1.217409, -2.668103, -0.826877, 1.570796, 1.655229],accel_mss,speed_ms,0,blend_radius_m)
    movel([0.085727, -1.216819, -2.668395, -0.827175, 1.570796, 1.656523],accel_mss,speed_ms,0,blend_radius_m)
    movel([0.085805, -1.215994, -2.668803, -0.827592, 1.570796, 1.656601],accel_mss,speed_ms,0,blend_radius_m)
    movel([0.085845, -1.215663, -2.668966, -0.827759, 1.570796, 1.656642],accel_mss,speed_ms,0,blend_radius_m)
    movel([0.085902, -1.215347, -2.669122, -0.827919, 1.570796, 1.656698],accel_mss,speed_ms,0,blend_radius_m)
    movel([0.086022, -1.214948, -2.669319, -0.828122, 1.570796, 1.656818],accel_mss,speed_ms,0,blend_radius_m)
    movel([0.086509, -1.214609, -2.669486, -0.828293, 1.570796, 1.657305],accel_mss,speed_ms,0,blend_radius_m)
    movel([0.087190, -1.214389, -2.669595, -0.828405, 1.570796, 1.657986],accel_mss,speed_ms,0,blend_radius_m)
    movel([0.087514, -1.214429, -2.669575, -0.828385, 1.570796, 1.658310],accel_mss,speed_ms,0,blend_radius_m)
    movel([0.087669, -1.214619, -2.669481, -0.828288, 1.570796, 1.658465],accel_mss,speed_ms,0,blend_radius_m)
    movel([0.087642, -1.214927, -2.669330, -0.828132, 1.570796, 1.658438],accel_mss,speed_ms,0,blend_radius_m)
    movel([0.087590, -1.215220, -2.669185, -0.827984, 1.570796, 1.658386],accel_mss,speed_ms,0,blend_radius_m)
    movel([0.087687, -1.215610, -2.668993, -0.827786, 1.570796, 1.658483],accel_mss,speed_ms,0,blend_radius_m)
    movel([0.087767, -1.215955, -2.668822, -0.827611, 1.570796, 1.658564],accel_mss,speed_ms,0,blend_radius_m)
    movel([0.088048, -1.216043, -2.668779, -0.827567, 1.570796, 1.658845],accel_mss,speed_ms,0,blend_radius_m)
    movel([0.088561, -1.216070, -2.668766, -0.827553, 1.570796, 1.659357],accel_mss,speed_ms,0,blend_radius_m)
    movel([0.088694, -1.216501, -2.668553, -0.827336, 1.570796, 1.659490],accel_mss,speed_ms,0,blend_radius_m)
    movel([0.088487, -1.216940, -2.668335, -0.827114, 1.570796, 1.659284],accel_mss,speed_ms,0,blend_radius_m)
    movel([0.088301, -1.217292, -2.668161, -0.826936, 1.570796, 1.659097],accel_mss,speed_ms,0,blend_radius_m)
    movel([0.088289, -1.217595, -2.668011, -0.826783, 1.570796, 1.659085],accel_mss,speed_ms,0,blend_radius_m)
    movel([0.088451, -1.217784, -2.667917, -0.826688, 1.570796, 1.659248],accel_mss,speed_ms,0,blend_radius_m)
    movel([0.088824, -1.218294, -2.667664, -0.826431, 1.570796, 1.659621],accel_mss,speed_ms,0,blend_radius_m)
    movel([0.089227, -1.219147, -2.667240, -0.826003, 1.570796, 1.660024],accel_mss,speed_ms,0,blend_radius_m)
    movel([0.089594, -1.220154, -2.666738, -0.825497, 1.570796, 1.660390],accel_mss,speed_ms,0,blend_radius_m)
    movel([0.089864, -1.221181, -2.666225, -0.824983, 1.570796, 1.660660],accel_mss,speed_ms,0,blend_radius_m)
    movel([0.090149, -1.222542, -2.665543, -0.824303, 1.570796, 1.660946],accel_mss,speed_ms,0,blend_radius_m)
    movel([0.090293, -1.223336, -2.665145, -0.823908, 1.570796, 1.661090],accel_mss,speed_ms,0,blend_radius_m)
    movel([0.090356, -1.223865, -2.664879, -0.823645, 1.570796, 1.661152],accel_mss,speed_ms,0,blend_radius_m)
    movel([0.090348, -1.224238, -2.664691, -0.823460, 1.570796, 1.661144],accel_mss,speed_ms,0,blend_radius_m)
    movel([0.090382, -1.224531, -2.664544, -0.823314, 1.570796, 1.661178],accel_mss,speed_ms,0,blend_radius_m)
    movel([0.090581, -1.224653, -2.664482, -0.823254, 1.570796, 1.661378],accel_mss,speed_ms,0,blend_radius_m)
    movel([0.090800, -1.224777, -2.664420, -0.823192, 1.570796, 1.661597],accel_mss,speed_ms,0,blend_radius_m)
    speed_ms = 0.003
    movel([0.090800, -1.228419, -2.666168, -0.817802, 1.570796, 1.661597],accel_mss,speed_ms,0,blend_radius_m)
    speed_ms = 0.007
    movel([0.090349, -1.228990, -2.665879, -0.817520, 1.570796, 1.661146],accel_mss,speed_ms,0,blend_radius_m)
    movel([0.089579, -1.229456, -2.665642, -0.817291, 1.570796, 1.660376],accel_mss,speed_ms,0,blend_radius_m)
    movel([0.088964, -1.229802, -2.665467, -0.817121, 1.570796, 1.659760],accel_mss,speed_ms,0,blend_radius_m)
    movel([0.087981, -1.230351, -2.665187, -0.816851, 1.570796, 1.658778],accel_mss,speed_ms,0,blend_radius_m)
    movel([0.086862, -1.230975, -2.664870, -0.816545, 1.570796, 1.657659],accel_mss,speed_ms,0,blend_radius_m)
    movel([0.085757, -1.231592, -2.664555, -0.816242, 1.570796, 1.656553],accel_mss,speed_ms,0,blend_radius_m)
    movel([0.084618, -1.232227, -2.664231, -0.815932, 1.570796, 1.655415],accel_mss,speed_ms,0,blend_radius_m)
    movel([0.083401, -1.232910, -2.663881, -0.815598, 1.570796, 1.654198],accel_mss,speed_ms,0,blend_radius_m)
    movel([0.082286, -1.233542, -2.663557, -0.815289, 1.570796, 1.653082],accel_mss,speed_ms,0,blend_radius_m)
    movel([0.081487, -1.233998, -2.663324, -0.815067, 1.570796, 1.652284],accel_mss,speed_ms,0,blend_radius_m)
    movel([0.077430, -1.236324, -2.662127, -0.813938, 1.570796, 1.648226],accel_mss,speed_ms,0,blend_radius_m)
    movel([0.075172, -1.237588, -2.661474, -0.813327, 1.570796, 1.645969],accel_mss,speed_ms,0,blend_radius_m)
    movel([0.073687, -1.238389, -2.661059, -0.812941, 1.570796, 1.644483],accel_mss,speed_ms,0,blend_radius_m)
    movel([0.073372, -1.238435, -2.661035, -0.812918, 1.570796, 1.644168],accel_mss,speed_ms,0,blend_radius_m)
    movel([0.073295, -1.238205, -2.661155, -0.813030, 1.570796, 1.644092],accel_mss,speed_ms,0,blend_radius_m)
    movel([0.073585, -1.237811, -2.661359, -0.813220, 1.570796, 1.644381],accel_mss,speed_ms,0,blend_radius_m)
    movel([0.073559, -1.237457, -2.661542, -0.813390, 1.570796, 1.644355],accel_mss,speed_ms,0,blend_radius_m)
    movel([0.073378, -1.237058, -2.661748, -0.813583, 1.570796, 1.644175],accel_mss,speed_ms,0,blend_radius_m)
    movel([0.073158, -1.235760, -2.662418, -0.814211, 1.570796, 1.643955],accel_mss,speed_ms,0,blend_radius_m)
    movel([0.072974, -1.234343, -2.663147, -0.814899, 1.570796, 1.643770],accel_mss,speed_ms,0,blend_radius_m)
    movel([0.072889, -1.233079, -2.663795, -0.815515, 1.570796, 1.643685],accel_mss,speed_ms,0,blend_radius_m)
    movel([0.072885, -1.232489, -2.664097, -0.815803, 1.570796, 1.643681],accel_mss,speed_ms,0,blend_radius_m)
    movel([0.072909, -1.231833, -2.664432, -0.816124, 1.570796, 1.643705],accel_mss,speed_ms,0,blend_radius_m)
    movel([0.072955, -1.231205, -2.664752, -0.816432, 1.570796, 1.643751],accel_mss,speed_ms,0,blend_radius_m)
    movel([0.073020, -1.230722, -2.664998, -0.816668, 1.570796, 1.643817],accel_mss,speed_ms,0,blend_radius_m)
    movel([0.073121, -1.230095, -2.665317, -0.816976, 1.570796, 1.643917],accel_mss,speed_ms,0,blend_radius_m)
    movel([0.073123, -1.229826, -2.665454, -0.817109, 1.570796, 1.643919],accel_mss,speed_ms,0,blend_radius_m)
    movel([0.072829, -1.229534, -2.665602, -0.817252, 1.570796, 1.643626],accel_mss,speed_ms,0,blend_radius_m)
    movel([0.072567, -1.229353, -2.665695, -0.817342, 1.570796, 1.643364],accel_mss,speed_ms,0,blend_radius_m)
    movel([0.072608, -1.228849, -2.665950, -0.817590, 1.570796, 1.643404],accel_mss,speed_ms,0,blend_radius_m)
    movel([0.072924, -1.228439, -2.666158, -0.817792, 1.570796, 1.643721],accel_mss,speed_ms,0,blend_radius_m)
    movel([0.073226, -1.228034, -2.666363, -0.817992, 1.570796, 1.644022],accel_mss,speed_ms,0,blend_radius_m)
    movel([0.073128, -1.227803, -2.666480, -0.818106, 1.570796, 1.643924],accel_mss,speed_ms,0,blend_radius_m)
    movel([0.073050, -1.227476, -2.666646, -0.818267, 1.570796, 1.643846],accel_mss,speed_ms,0,blend_radius_m)
    movel([0.072942, -1.227155, -2.666808, -0.818426, 1.570796, 1.643738],accel_mss,speed_ms,0,blend_radius_m)
    movel([0.072715, -1.226995, -2.666888, -0.818505, 1.570796, 1.643512],accel_mss,speed_ms,0,blend_radius_m)
    movel([0.072769, -1.226616, -2.667080, -0.818693, 1.570796, 1.643566],accel_mss,speed_ms,0,blend_radius_m)
    movel([0.073235, -1.226064, -2.667358, -0.818967, 1.570796, 1.644032],accel_mss,speed_ms,0,blend_radius_m)
    movel([0.073730, -1.225528, -2.667628, -0.819233, 1.570796, 1.644526],accel_mss,speed_ms,0,blend_radius_m)
    movel([0.074179, -1.225331, -2.667727, -0.819331, 1.570796, 1.644975],accel_mss,speed_ms,0,blend_radius_m)
    movel([0.074415, -1.225409, -2.667688, -0.819292, 1.570796, 1.645212],accel_mss,speed_ms,0,blend_radius_m)
    movel([0.074609, -1.225538, -2.667623, -0.819228, 1.570796, 1.645406],accel_mss,speed_ms,0,blend_radius_m)
    movel([0.074697, -1.225922, -2.667430, -0.819037, 1.570796, 1.645493],accel_mss,speed_ms,0,blend_radius_m)
    movel([0.074870, -1.226198, -2.667291, -0.818900, 1.570796, 1.645666],accel_mss,speed_ms,0,blend_radius_m)
    movel([0.075082, -1.226424, -2.667177, -0.818788, 1.570796, 1.645878],accel_mss,speed_ms,0,blend_radius_m)
    movel([0.075630, -1.226227, -2.667276, -0.818886, 1.570796, 1.646426],accel_mss,speed_ms,0,blend_radius_m)
    movel([0.076550, -1.225573, -2.667606, -0.819211, 1.570796, 1.647346],accel_mss,speed_ms,0,blend_radius_m)
    movel([0.077489, -1.224883, -2.667953, -0.819554, 1.570796, 1.648285],accel_mss,speed_ms,0,blend_radius_m)
    movel([0.077732, -1.224573, -2.668108, -0.819708, 1.570796, 1.648528],accel_mss,speed_ms,0,blend_radius_m)
    movel([0.077653, -1.224307, -2.668242, -0.819840, 1.570796, 1.648449],accel_mss,speed_ms,0,blend_radius_m)
    movel([0.077678, -1.223945, -2.668423, -0.820020, 1.570796, 1.648474],accel_mss,speed_ms,0,blend_radius_m)
    movel([0.077699, -1.223674, -2.668559, -0.820155, 1.570796, 1.648495],accel_mss,speed_ms,0,blend_radius_m)
    movel([0.077413, -1.223292, -2.668751, -0.820346, 1.570796, 1.648209],accel_mss,speed_ms,0,blend_radius_m)
    movel([0.077317, -1.222840, -2.668977, -0.820572, 1.570796, 1.648113],accel_mss,speed_ms,0,blend_radius_m)
    movel([0.077299, -1.222333, -2.669230, -0.820825, 1.570796, 1.648095],accel_mss,speed_ms,0,blend_radius_m)
    movel([0.077389, -1.221932, -2.669431, -0.821026, 1.570796, 1.648186],accel_mss,speed_ms,0,blend_radius_m)
    movel([0.077615, -1.221557, -2.669618, -0.821214, 1.570796, 1.648412],accel_mss,speed_ms,0,blend_radius_m)
    movel([0.078010, -1.221162, -2.669815, -0.821412, 1.570796, 1.648807],accel_mss,speed_ms,0,blend_radius_m)
    movel([0.078613, -1.220713, -2.670038, -0.821637, 1.570796, 1.649409],accel_mss,speed_ms,0,blend_radius_m)
    movel([0.079495, -1.220163, -2.670312, -0.821914, 1.570796, 1.650291],accel_mss,speed_ms,0,blend_radius_m)
    movel([0.080567, -1.219561, -2.670611, -0.822217, 1.570796, 1.651364],accel_mss,speed_ms,0,blend_radius_m)
    movel([0.081345, -1.219203, -2.670789, -0.822398, 1.570796, 1.652142],accel_mss,speed_ms,0,blend_radius_m)
    movel([0.081899, -1.219048, -2.670866, -0.822475, 1.570796, 1.652696],accel_mss,speed_ms,0,blend_radius_m)
    movel([0.082256, -1.219095, -2.670842, -0.822452, 1.570796, 1.653053],accel_mss,speed_ms,0,blend_radius_m)
    movel([0.082498, -1.219340, -2.670721, -0.822328, 1.570796, 1.653294],accel_mss,speed_ms,0,blend_radius_m)
    movel([0.082652, -1.219772, -2.670506, -0.822111, 1.570796, 1.653448],accel_mss,speed_ms,0,blend_radius_m)
    movel([0.082703, -1.220236, -2.670276, -0.821877, 1.570796, 1.653499],accel_mss,speed_ms,0,blend_radius_m)
    movel([0.082589, -1.220578, -2.670105, -0.821705, 1.570796, 1.653386],accel_mss,speed_ms,0,blend_radius_m)
    movel([0.082550, -1.220971, -2.669910, -0.821508, 1.570796, 1.653347],accel_mss,speed_ms,0,blend_radius_m)
    movel([0.082765, -1.221186, -2.669803, -0.821400, 1.570796, 1.653561],accel_mss,speed_ms,0,blend_radius_m)
    movel([0.082850, -1.221412, -2.669690, -0.821287, 1.570796, 1.653646],accel_mss,speed_ms,0,blend_radius_m)
    movel([0.083106, -1.221582, -2.669605, -0.821202, 1.570796, 1.653902],accel_mss,speed_ms,0,blend_radius_m)
    movel([0.083419, -1.221488, -2.669652, -0.821249, 1.570796, 1.654215],accel_mss,speed_ms,0,blend_radius_m)
    movel([0.083853, -1.221318, -2.669737, -0.821334, 1.570796, 1.654650],accel_mss,speed_ms,0,blend_radius_m)
    movel([0.084433, -1.221063, -2.669864, -0.821462, 1.570796, 1.655229],accel_mss,speed_ms,0,blend_radius_m)
    movel([0.085727, -1.220473, -2.670158, -0.821758, 1.570796, 1.656523],accel_mss,speed_ms,0,blend_radius_m)
    movel([0.085805, -1.219650, -2.670567, -0.822172, 1.570796, 1.656601],accel_mss,speed_ms,0,blend_radius_m)
    movel([0.085845, -1.219319, -2.670731, -0.822339, 1.570796, 1.656642],accel_mss,speed_ms,0,blend_radius_m)
    movel([0.085902, -1.219004, -2.670887, -0.822498, 1.570796, 1.656698],accel_mss,speed_ms,0,blend_radius_m)
    movel([0.086022, -1.218605, -2.671085, -0.822699, 1.570796, 1.656818],accel_mss,speed_ms,0,blend_radius_m)
    movel([0.086509, -1.218267, -2.671253, -0.822870, 1.570796, 1.657305],accel_mss,speed_ms,0,blend_radius_m)
    movel([0.087190, -1.218047, -2.671361, -0.822981, 1.570796, 1.657986],accel_mss,speed_ms,0,blend_radius_m)
    movel([0.087514, -1.218087, -2.671342, -0.822960, 1.570796, 1.658310],accel_mss,speed_ms,0,blend_radius_m)
    movel([0.087669, -1.218277, -2.671248, -0.822865, 1.570796, 1.658465],accel_mss,speed_ms,0,blend_radius_m)
    movel([0.087642, -1.218584, -2.671096, -0.822710, 1.570796, 1.658438],accel_mss,speed_ms,0,blend_radius_m)
    movel([0.087590, -1.218877, -2.670950, -0.822562, 1.570796, 1.658386],accel_mss,speed_ms,0,blend_radius_m)
    movel([0.087687, -1.219266, -2.670758, -0.822366, 1.570796, 1.658483],accel_mss,speed_ms,0,blend_radius_m)
    movel([0.087767, -1.219611, -2.670586, -0.822192, 1.570796, 1.658564],accel_mss,speed_ms,0,blend_radius_m)
    movel([0.088048, -1.219699, -2.670543, -0.822148, 1.570796, 1.658845],accel_mss,speed_ms,0,blend_radius_m)
    movel([0.088561, -1.219725, -2.670529, -0.822134, 1.570796, 1.659357],accel_mss,speed_ms,0,blend_radius_m)
    movel([0.088694, -1.220156, -2.670316, -0.821918, 1.570796, 1.659490],accel_mss,speed_ms,0,blend_radius_m)
    movel([0.088487, -1.220594, -2.670098, -0.821697, 1.570796, 1.659284],accel_mss,speed_ms,0,blend_radius_m)
    movel([0.088301, -1.220945, -2.669923, -0.821521, 1.570796, 1.659097],accel_mss,speed_ms,0,blend_radius_m)
    movel([0.088289, -1.221248, -2.669772, -0.821369, 1.570796, 1.659085],accel_mss,speed_ms,0,blend_radius_m)
    movel([0.088451, -1.221437, -2.669678, -0.821275, 1.570796, 1.659248],accel_mss,speed_ms,0,blend_radius_m)
    movel([0.088824, -1.221946, -2.669424, -0.821019, 1.570796, 1.659621],accel_mss,speed_ms,0,blend_radius_m)
    movel([0.089227, -1.222797, -2.668998, -0.820593, 1.570796, 1.660024],accel_mss,speed_ms,0,blend_radius_m)
    movel([0.089594, -1.223803, -2.668495, -0.820091, 1.570796, 1.660390],accel_mss,speed_ms,0,blend_radius_m)
    movel([0.089864, -1.224829, -2.667980, -0.819581, 1.570796, 1.660660],accel_mss,speed_ms,0,blend_radius_m)
    movel([0.090149, -1.226188, -2.667296, -0.818905, 1.570796, 1.660946],accel_mss,speed_ms,0,blend_radius_m)
    movel([0.090293, -1.226980, -2.666896, -0.818513, 1.570796, 1.661090],accel_mss,speed_ms,0,blend_radius_m)
    movel([0.090356, -1.227508, -2.666629, -0.818252, 1.570796, 1.661152],accel_mss,speed_ms,0,blend_radius_m)
    movel([0.090348, -1.227880, -2.666441, -0.818068, 1.570796, 1.661144],accel_mss,speed_ms,0,blend_radius_m)
    movel([0.090382, -1.228173, -2.666293, -0.817923, 1.570796, 1.661178],accel_mss,speed_ms,0,blend_radius_m)
    movel([0.090581, -1.228294, -2.666231, -0.817863, 1.570796, 1.661378],accel_mss,speed_ms,0,blend_radius_m)
    movel([0.090800, -1.228419, -2.666168, -0.817802, 1.570796, 1.661597],accel_mss,speed_ms,0,blend_radius_m)
    speed_ms = 0.003
    movel([0.090800, -1.214052, -2.659125, -0.839212, 1.570796, 1.661597],accel_mss,speed_ms,0,blend_radius_m)
    speed_ms = 1.000
    movel([0.090800, -1.186880, -2.644666, -0.880842, 1.570796, 1.661597],accel_mss,speed_ms,0,blend_radius_m)
    movel([0.087310, -1.181711, -2.647130, -0.883548, 1.570796, 1.658107],accel_mss,speed_ms,0,blend_radius_m)
    movel([0.087310, -1.208926, -2.661656, -0.841806, 1.570796, 1.658107],accel_mss,speed_ms,0,blend_radius_m)
    speed_ms = 0.003
    movel([0.087310, -1.219674, -2.666977, -0.825738, 1.570796, 1.658107],accel_mss,speed_ms,0,blend_radius_m)
    speed_ms = 0.007
    movel([0.086870, -1.219855, -2.666887, -0.825647, 1.570796, 1.657666],accel_mss,speed_ms,0,blend_radius_m)
    movel([0.086396, -1.219968, -2.666831, -0.825590, 1.570796, 1.657192],accel_mss,speed_ms,0,blend_radius_m)
    movel([0.086386, -1.219703, -2.666963, -0.825723, 1.570796, 1.657182],accel_mss,speed_ms,0,blend_radius_m)
    movel([0.086847, -1.219492, -2.667068, -0.825829, 1.570796, 1.657643],accel_mss,speed_ms,0,blend_radius_m)
    movel([0.087324, -1.219355, -2.667136, -0.825898, 1.570796, 1.658120],accel_mss,speed_ms,0,blend_radius_m)
    movel([0.087401, -1.219581, -2.667023, -0.825784, 1.570796, 1.658197],accel_mss,speed_ms,0,blend_radius_m)
    speed_ms = 0.003
    movel([0.087310, -1.223324, -2.668735, -0.820331, 1.570796, 1.658107],accel_mss,speed_ms,0,blend_radius_m)
    speed_ms = 0.007
    movel([0.086870, -1.223505, -2.668644, -0.820240, 1.570796, 1.657666],accel_mss,speed_ms,0,blend_radius_m)
    movel([0.086396, -1.223617, -2.668588, -0.820184, 1.570796, 1.657192],accel_mss,speed_ms,0,blend_radius_m)
    movel([0.086386, -1.223352, -2.668720, -0.820316, 1.570796, 1.657182],accel_mss,speed_ms,0,blend_radius_m)
    movel([0.086847, -1.223142, -2.668826, -0.820421, 1.570796, 1.657643],accel_mss,speed_ms,0,blend_radius_m)
    movel([0.087324, -1.223005, -2.668894, -0.820489, 1.570796, 1.658120],accel_mss,speed_ms,0,blend_radius_m)
    movel([0.087401, -1.223231, -2.668781, -0.820377, 1.570796, 1.658197],accel_mss,speed_ms,0,blend_radius_m)
    speed_ms = 0.003
    movel([0.087310, -1.208926, -2.661656, -0.841806, 1.570796, 1.658107],accel_mss,speed_ms,0,blend_radius_m)
    speed_ms = 1.000
    movel([0.087310, -1.181711, -2.647130, -0.883548, 1.570796, 1.658107],accel_mss,speed_ms,0,blend_radius_m)
    movel([0.082030, -1.179475, -2.648187, -0.884727, 1.570796, 1.652827],accel_mss,speed_ms,0,blend_radius_m)
    movel([0.082030, -1.206709, -2.662743, -0.842937, 1.570796, 1.652827],accel_mss,speed_ms,0,blend_radius_m)
    speed_ms = 0.003
    movel([0.082030, -1.217466, -2.668075, -0.826848, 1.570796, 1.652827],accel_mss,speed_ms,0,blend_radius_m)
    speed_ms = 0.007
    movel([0.081697, -1.217749, -2.667934, -0.826706, 1.570796, 1.652493],accel_mss,speed_ms,0,blend_radius_m)
    movel([0.080452, -1.218501, -2.667561, -0.826327, 1.570796, 1.651249],accel_mss,speed_ms,0,blend_radius_m)
    movel([0.079236, -1.219205, -2.667211, -0.825973, 1.570796, 1.650033],accel_mss,speed_ms,0,blend_radius_m)
    movel([0.078580, -1.219519, -2.667054, -0.825816, 1.570796, 1.649376],accel_mss,speed_ms,0,blend_radius_m)
    movel([0.078178, -1.219588, -2.667020, -0.825781, 1.570796, 1.648975],accel_mss,speed_ms,0,blend_radius_m)
    movel([0.078075, -1.219125, -2.667250, -0.826013, 1.570796, 1.648872],accel_mss,speed_ms,0,blend_radius_m)
    movel([0.078079, -1.218647, -2.667489, -0.826254, 1.570796, 1.648875],accel_mss,speed_ms,0,blend_radius_m)
    movel([0.078144, -1.218302, -2.667660, -0.826427, 1.570796, 1.648940],accel_mss,speed_ms,0,blend_radius_m)
    movel([0.078358, -1.217999, -2.667810, -0.826580, 1.570796, 1.649154],accel_mss,speed_ms,0,blend_radius_m)
    movel([0.078770, -1.217643, -2.667987, -0.826759, 1.570796, 1.649567],accel_mss,speed_ms,0,blend_radius_m)
    movel([0.079360, -1.217236, -2.668189, -0.826965, 1.570796, 1.650157],accel_mss,speed_ms,0,blend_radius_m)
    movel([0.080137, -1.216785, -2.668412, -0.827192, 1.570796, 1.650933],accel_mss,speed_ms,0,blend_radius_m)
    movel([0.080944, -1.216386, -2.668609, -0.827394, 1.570796, 1.651740],accel_mss,speed_ms,0,blend_radius_m)
    movel([0.081471, -1.216237, -2.668683, -0.827469, 1.570796, 1.652267],accel_mss,speed_ms,0,blend_radius_m)
    movel([0.081790, -1.216308, -2.668648, -0.827433, 1.570796, 1.652586],accel_mss,speed_ms,0,blend_radius_m)
    movel([0.081946, -1.216589, -2.668509, -0.827291, 1.570796, 1.652742],accel_mss,speed_ms,0,blend_radius_m)
    movel([0.082016, -1.216879, -2.668365, -0.827144, 1.570796, 1.652813],accel_mss,speed_ms,0,blend_radius_m)
    movel([0.082108, -1.217092, -2.668260, -0.827037, 1.570796, 1.652905],accel_mss,speed_ms,0,blend_radius_m)
    movel([0.082098, -1.217366, -2.668124, -0.826899, 1.570796, 1.652894],accel_mss,speed_ms,0,blend_radius_m)
    speed_ms = 0.003
    movel([0.082030, -1.221119, -2.669836, -0.821434, 1.570796, 1.652827],accel_mss,speed_ms,0,blend_radius_m)
    speed_ms = 0.007
    movel([0.081697, -1.221401, -2.669695, -0.821292, 1.570796, 1.652493],accel_mss,speed_ms,0,blend_radius_m)
    movel([0.080452, -1.222152, -2.669321, -0.820916, 1.570796, 1.651249],accel_mss,speed_ms,0,blend_radius_m)
    movel([0.079236, -1.222856, -2.668969, -0.820564, 1.570796, 1.650033],accel_mss,speed_ms,0,blend_radius_m)
    movel([0.078580, -1.223169, -2.668812, -0.820408, 1.570796, 1.649376],accel_mss,speed_ms,0,blend_radius_m)
    movel([0.078178, -1.223238, -2.668778, -0.820373, 1.570796, 1.648975],accel_mss,speed_ms,0,blend_radius_m)
    movel([0.078075, -1.222776, -2.669009, -0.820604, 1.570796, 1.648872],accel_mss,speed_ms,0,blend_radius_m)
    movel([0.078079, -1.222298, -2.669248, -0.820843, 1.570796, 1.648875],accel_mss,speed_ms,0,blend_radius_m)
    movel([0.078144, -1.221954, -2.669420, -0.821015, 1.570796, 1.648940],accel_mss,speed_ms,0,blend_radius_m)
    movel([0.078358, -1.221652, -2.669571, -0.821167, 1.570796, 1.649154],accel_mss,speed_ms,0,blend_radius_m)
    movel([0.078770, -1.221296, -2.669748, -0.821345, 1.570796, 1.649567],accel_mss,speed_ms,0,blend_radius_m)
    movel([0.079360, -1.220889, -2.669951, -0.821549, 1.570796, 1.650157],accel_mss,speed_ms,0,blend_radius_m)
    movel([0.080137, -1.220439, -2.670175, -0.821775, 1.570796, 1.650933],accel_mss,speed_ms,0,blend_radius_m)
    movel([0.080944, -1.220041, -2.670373, -0.821976, 1.570796, 1.651740],accel_mss,speed_ms,0,blend_radius_m)
    movel([0.081471, -1.219892, -2.670447, -0.822051, 1.570796, 1.652267],accel_mss,speed_ms,0,blend_radius_m)
    movel([0.081790, -1.219963, -2.670411, -0.822014, 1.570796, 1.652586],accel_mss,speed_ms,0,blend_radius_m)
    movel([0.081946, -1.220244, -2.670272, -0.821874, 1.570796, 1.652742],accel_mss,speed_ms,0,blend_radius_m)
    movel([0.082016, -1.220533, -2.670128, -0.821728, 1.570796, 1.652813],accel_mss,speed_ms,0,blend_radius_m)
    movel([0.082108, -1.220746, -2.670022, -0.821621, 1.570796, 1.652905],accel_mss,speed_ms,0,blend_radius_m)
    movel([0.082098, -1.221019, -2.669886, -0.821484, 1.570796, 1.652894],accel_mss,speed_ms,0,blend_radius_m)
    speed_ms = 0.003
    movel([0.082030, -1.206709, -2.662743, -0.842937, 1.570796, 1.652827],accel_mss,speed_ms,0,blend_radius_m)
    speed_ms = 1.000
    movel([0.082030, -1.179475, -2.648187, -0.884727, 1.570796, 1.652827],accel_mss,speed_ms,0,blend_radius_m)
    movel([0.076474, -1.187386, -2.644424, -0.880579, 1.570796, 1.647270],accel_mss,speed_ms,0,blend_radius_m)
    movel([0.076474, -1.214553, -2.658876, -0.838960, 1.570796, 1.647270],accel_mss,speed_ms,0,blend_radius_m)
    speed_ms = 0.003
    movel([0.076474, -1.225276, -2.664168, -0.822945, 1.570796, 1.647270],accel_mss,speed_ms,0,blend_radius_m)
    speed_ms = 0.007
    movel([0.076414, -1.225602, -2.664003, -0.822783, 1.570796, 1.647210],accel_mss,speed_ms,0,blend_radius_m)
    movel([0.076013, -1.225935, -2.663835, -0.822619, 1.570796, 1.646810],accel_mss,speed_ms,0,blend_radius_m)
    movel([0.075745, -1.226284, -2.663659, -0.822446, 1.570796, 1.646542],accel_mss,speed_ms,0,blend_radius_m)
    movel([0.075688, -1.226656, -2.663470, -0.822263, 1.570796, 1.646484],accel_mss,speed_ms,0,blend_radius_m)
    movel([0.075585, -1.227082, -2.663255, -0.822053, 1.570796, 1.646381],accel_mss,speed_ms,0,blend_radius_m)
    movel([0.075278, -1.227242, -2.663174, -0.821973, 1.570796, 1.646074],accel_mss,speed_ms,0,blend_radius_m)
    movel([0.075133, -1.227069, -2.663261, -0.822059, 1.570796, 1.645929],accel_mss,speed_ms,0,blend_radius_m)
    movel([0.074972, -1.226910, -2.663342, -0.822137, 1.570796, 1.645768],accel_mss,speed_ms,0,blend_radius_m)
    movel([0.074300, -1.227259, -2.663165, -0.821965, 1.570796, 1.645096],accel_mss,speed_ms,0,blend_radius_m)
    movel([0.073968, -1.227370, -2.663109, -0.821910, 1.570796, 1.644764],accel_mss,speed_ms,0,blend_radius_m)
    movel([0.074075, -1.226987, -2.663303, -0.822099, 1.570796, 1.644872],accel_mss,speed_ms,0,blend_radius_m)
    movel([0.074398, -1.226677, -2.663460, -0.822252, 1.570796, 1.645194],accel_mss,speed_ms,0,blend_radius_m)
    movel([0.074745, -1.226346, -2.663627, -0.822416, 1.570796, 1.645542],accel_mss,speed_ms,0,blend_radius_m)
    movel([0.074798, -1.226034, -2.663785, -0.822570, 1.570796, 1.645594],accel_mss,speed_ms,0,blend_radius_m)
    movel([0.074884, -1.225697, -2.663955, -0.822736, 1.570796, 1.645680],accel_mss,speed_ms,0,blend_radius_m)
    movel([0.075260, -1.225619, -2.663995, -0.822775, 1.570796, 1.646057],accel_mss,speed_ms,0,blend_radius_m)
    movel([0.075513, -1.225654, -2.663977, -0.822758, 1.570796, 1.646310],accel_mss,speed_ms,0,blend_radius_m)
    movel([0.075891, -1.225492, -2.664059, -0.822838, 1.570796, 1.646687],accel_mss,speed_ms,0,blend_radius_m)
    movel([0.076264, -1.225319, -2.664146, -0.822924, 1.570796, 1.647060],accel_mss,speed_ms,0,blend_radius_m)
    speed_ms = 0.003
    movel([0.076474, -1.228917, -2.665916, -0.817556, 1.570796, 1.647270],accel_mss,speed_ms,0,blend_radius_m)
    speed_ms = 0.007
    movel([0.076414, -1.229243, -2.665751, -0.817396, 1.570796, 1.647210],accel_mss,speed_ms,0,blend_radius_m)
    movel([0.076013, -1.229575, -2.665582, -0.817232, 1.570796, 1.646810],accel_mss,speed_ms,0,blend_radius_m)
    movel([0.075745, -1.229923, -2.665405, -0.817061, 1.570796, 1.646542],accel_mss,speed_ms,0,blend_radius_m)
    movel([0.075688, -1.230294, -2.665216, -0.816879, 1.570796, 1.646484],accel_mss,speed_ms,0,blend_radius_m)
    movel([0.075585, -1.230719, -2.665000, -0.816670, 1.570796, 1.646381],accel_mss,speed_ms,0,blend_radius_m)
    movel([0.075278, -1.230879, -2.664918, -0.816591, 1.570796, 1.646074],accel_mss,speed_ms,0,blend_radius_m)
    movel([0.075133, -1.230707, -2.665006, -0.816676, 1.570796, 1.645929],accel_mss,speed_ms,0,blend_radius_m)
    movel([0.074972, -1.230548, -2.665087, -0.816754, 1.570796, 1.645768],accel_mss,speed_ms,0,blend_radius_m)
    movel([0.074300, -1.230897, -2.664909, -0.816583, 1.570796, 1.645096],accel_mss,speed_ms,0,blend_radius_m)
    movel([0.073968, -1.231007, -2.664853, -0.816529, 1.570796, 1.644764],accel_mss,speed_ms,0,blend_radius_m)
    movel([0.074075, -1.230625, -2.665048, -0.816716, 1.570796, 1.644872],accel_mss,speed_ms,0,blend_radius_m)
    movel([0.074398, -1.230315, -2.665206, -0.816868, 1.570796, 1.645194],accel_mss,speed_ms,0,blend_radius_m)
    movel([0.074745, -1.229985, -2.665373, -0.817031, 1.570796, 1.645542],accel_mss,speed_ms,0,blend_radius_m)
    movel([0.074798, -1.229673, -2.665532, -0.817184, 1.570796, 1.645594],accel_mss,speed_ms,0,blend_radius_m)
    movel([0.074884, -1.229337, -2.665702, -0.817349, 1.570796, 1.645680],accel_mss,speed_ms,0,blend_radius_m)
    movel([0.075260, -1.229259, -2.665742, -0.817388, 1.570796, 1.646057],accel_mss,speed_ms,0,blend_radius_m)
    movel([0.075513, -1.229294, -2.665725, -0.817370, 1.570796, 1.646310],accel_mss,speed_ms,0,blend_radius_m)
    movel([0.075891, -1.229132, -2.665807, -0.817450, 1.570796, 1.646687],accel_mss,speed_ms,0,blend_radius_m)
    movel([0.076264, -1.228959, -2.665894, -0.817535, 1.570796, 1.647060],accel_mss,speed_ms,0,blend_radius_m)
    speed_ms = 0.003
    movel([0.076474, -1.214553, -2.658876, -0.838960, 1.570796, 1.647270],accel_mss,speed_ms,0,blend_radius_m)
    speed_ms = 1.000
    movel([0.076474, -1.187386, -2.644424, -0.880579, 1.570796, 1.647270],accel_mss,speed_ms,0,blend_radius_m)
    movel([0.079801, -1.186394, -2.644900, -0.881096, 1.570796, 1.650597],accel_mss,speed_ms,0,blend_radius_m)
    movel([0.079801, -1.213569, -2.659364, -0.839455, 1.570796, 1.650597],accel_mss,speed_ms,0,blend_radius_m)
    speed_ms = 0.003
    movel([0.079801, -1.224297, -2.664662, -0.823431, 1.570796, 1.650597],accel_mss,speed_ms,0,blend_radius_m)
    speed_ms = 0.007
    movel([0.079957, -1.223750, -2.664937, -0.823702, 1.570796, 1.650754],accel_mss,speed_ms,0,blend_radius_m)
    movel([0.080112, -1.223252, -2.665187, -0.823950, 1.570796, 1.650909],accel_mss,speed_ms,0,blend_radius_m)
    movel([0.080251, -1.222837, -2.665395, -0.824157, 1.570796, 1.651048],accel_mss,speed_ms,0,blend_radius_m)
    movel([0.080545, -1.222482, -2.665573, -0.824333, 1.570796, 1.651342],accel_mss,speed_ms,0,blend_radius_m)
    movel([0.081160, -1.222096, -2.665767, -0.824526, 1.570796, 1.651957],accel_mss,speed_ms,0,blend_radius_m)
    movel([0.081785, -1.221737, -2.665947, -0.824705, 1.570796, 1.652581],accel_mss,speed_ms,0,blend_radius_m)
    movel([0.081963, -1.221989, -2.665821, -0.824579, 1.570796, 1.652759],accel_mss,speed_ms,0,blend_radius_m)
    movel([0.081869, -1.222314, -2.665658, -0.824417, 1.570796, 1.652665],accel_mss,speed_ms,0,blend_radius_m)
    movel([0.081742, -1.222691, -2.665469, -0.824229, 1.570796, 1.652538],accel_mss,speed_ms,0,blend_radius_m)
    movel([0.081390, -1.223678, -2.664973, -0.823738, 1.570796, 1.652186],accel_mss,speed_ms,0,blend_radius_m)
    movel([0.081936, -1.223554, -2.665035, -0.823800, 1.570796, 1.652733],accel_mss,speed_ms,0,blend_radius_m)
    movel([0.082357, -1.223471, -2.665077, -0.823841, 1.570796, 1.653153],accel_mss,speed_ms,0,blend_radius_m)
    movel([0.082633, -1.223473, -2.665076, -0.823840, 1.570796, 1.653430],accel_mss,speed_ms,0,blend_radius_m)
    movel([0.082552, -1.223879, -2.664872, -0.823638, 1.570796, 1.653349],accel_mss,speed_ms,0,blend_radius_m)
    movel([0.082407, -1.224259, -2.664681, -0.823449, 1.570796, 1.653203],accel_mss,speed_ms,0,blend_radius_m)
    movel([0.082235, -1.224712, -2.664452, -0.823225, 1.570796, 1.653031],accel_mss,speed_ms,0,blend_radius_m)
    movel([0.082051, -1.225198, -2.664207, -0.822984, 1.570796, 1.652847],accel_mss,speed_ms,0,blend_radius_m)
    movel([0.081855, -1.225722, -2.663943, -0.822724, 1.570796, 1.652651],accel_mss,speed_ms,0,blend_radius_m)
    movel([0.081649, -1.226292, -2.663655, -0.822442, 1.570796, 1.652446],accel_mss,speed_ms,0,blend_radius_m)
    movel([0.081465, -1.226816, -2.663389, -0.822184, 1.570796, 1.652262],accel_mss,speed_ms,0,blend_radius_m)
    movel([0.081341, -1.227200, -2.663195, -0.821994, 1.570796, 1.652137],accel_mss,speed_ms,0,blend_radius_m)
    movel([0.081235, -1.227506, -2.663040, -0.821843, 1.570796, 1.652031],accel_mss,speed_ms,0,blend_radius_m)
    movel([0.081014, -1.228020, -2.662779, -0.821590, 1.570796, 1.651811],accel_mss,speed_ms,0,blend_radius_m)
    movel([0.080629, -1.228055, -2.662761, -0.821573, 1.570796, 1.651425],accel_mss,speed_ms,0,blend_radius_m)
    movel([0.080637, -1.227615, -2.662984, -0.821790, 1.570796, 1.651433],accel_mss,speed_ms,0,blend_radius_m)
    movel([0.080778, -1.226782, -2.663407, -0.822201, 1.570796, 1.651575],accel_mss,speed_ms,0,blend_radius_m)
    movel([0.080941, -1.225848, -2.663879, -0.822662, 1.570796, 1.651737],accel_mss,speed_ms,0,blend_radius_m)
    movel([0.080916, -1.225513, -2.664048, -0.822828, 1.570796, 1.651712],accel_mss,speed_ms,0,blend_radius_m)
    movel([0.080357, -1.225662, -2.663973, -0.822754, 1.570796, 1.651153],accel_mss,speed_ms,0,blend_radius_m)
    movel([0.079985, -1.225891, -2.663857, -0.822641, 1.570796, 1.650781],accel_mss,speed_ms,0,blend_radius_m)
    movel([0.079609, -1.226069, -2.663767, -0.822552, 1.570796, 1.650405],accel_mss,speed_ms,0,blend_radius_m)
    movel([0.079304, -1.226069, -2.663767, -0.822553, 1.570796, 1.650100],accel_mss,speed_ms,0,blend_radius_m)
    movel([0.079388, -1.225778, -2.663914, -0.822696, 1.570796, 1.650184],accel_mss,speed_ms,0,blend_radius_m)
    movel([0.079510, -1.225353, -2.664129, -0.822907, 1.570796, 1.650306],accel_mss,speed_ms,0,blend_radius_m)
    movel([0.079650, -1.224846, -2.664385, -0.823158, 1.570796, 1.650447],accel_mss,speed_ms,0,blend_radius_m)
    movel([0.079801, -1.224297, -2.664662, -0.823431, 1.570796, 1.650597],accel_mss,speed_ms,0,blend_radius_m)
    speed_ms = 0.003
    movel([0.079801, -1.227939, -2.666411, -0.818039, 1.570796, 1.650597],accel_mss,speed_ms,0,blend_radius_m)
    speed_ms = 0.007
    movel([0.079957, -1.227393, -2.666688, -0.818309, 1.570796, 1.650754],accel_mss,speed_ms,0,blend_radius_m)
    movel([0.080112, -1.226896, -2.666938, -0.818554, 1.570796, 1.650909],accel_mss,speed_ms,0,blend_radius_m)
    movel([0.080251, -1.226482, -2.667148, -0.818760, 1.570796, 1.651048],accel_mss,speed_ms,0,blend_radius_m)
    movel([0.080545, -1.226128, -2.667326, -0.818935, 1.570796, 1.651342],accel_mss,speed_ms,0,blend_radius_m)
    movel([0.081160, -1.225741, -2.667521, -0.819127, 1.570796, 1.651957],accel_mss,speed_ms,0,blend_radius_m)
    movel([0.081785, -1.225383, -2.667701, -0.819305, 1.570796, 1.652581],accel_mss,speed_ms,0,blend_radius_m)
    movel([0.081963, -1.225635, -2.667574, -0.819180, 1.570796, 1.652759],accel_mss,speed_ms,0,blend_radius_m)
    movel([0.081869, -1.225959, -2.667411, -0.819019, 1.570796, 1.652665],accel_mss,speed_ms,0,blend_radius_m)
    movel([0.081742, -1.226335, -2.667221, -0.818832, 1.570796, 1.652538],accel_mss,speed_ms,0,blend_radius_m)
    movel([0.081390, -1.227321, -2.666724, -0.818344, 1.570796, 1.652186],accel_mss,speed_ms,0,blend_radius_m)
    movel([0.081936, -1.227198, -2.666786, -0.818405, 1.570796, 1.652733],accel_mss,speed_ms,0,blend_radius_m)
    movel([0.082357, -1.227115, -2.666828, -0.818446, 1.570796, 1.653153],accel_mss,speed_ms,0,blend_radius_m)
    movel([0.082633, -1.227117, -2.666827, -0.818445, 1.570796, 1.653430],accel_mss,speed_ms,0,blend_radius_m)
    movel([0.082552, -1.227521, -2.666623, -0.818245, 1.570796, 1.653349],accel_mss,speed_ms,0,blend_radius_m)
    movel([0.082407, -1.227901, -2.666430, -0.818057, 1.570796, 1.653203],accel_mss,speed_ms,0,blend_radius_m)
    movel([0.082235, -1.228354, -2.666201, -0.817834, 1.570796, 1.653031],accel_mss,speed_ms,0,blend_radius_m)
    movel([0.082051, -1.228839, -2.665955, -0.817595, 1.570796, 1.652847],accel_mss,speed_ms,0,blend_radius_m)
    movel([0.081855, -1.229362, -2.665690, -0.817337, 1.570796, 1.652651],accel_mss,speed_ms,0,blend_radius_m)
    movel([0.081649, -1.229931, -2.665401, -0.817057, 1.570796, 1.652446],accel_mss,speed_ms,0,blend_radius_m)
    movel([0.081465, -1.230454, -2.665135, -0.816800, 1.570796, 1.652262],accel_mss,speed_ms,0,blend_radius_m)
    movel([0.081341, -1.230837, -2.664940, -0.816612, 1.570796, 1.652137],accel_mss,speed_ms,0,blend_radius_m)
    movel([0.081235, -1.231143, -2.664784, -0.816462, 1.570796, 1.652031],accel_mss,speed_ms,0,blend_radius_m)
    movel([0.081014, -1.231656, -2.664522, -0.816211, 1.570796, 1.651811],accel_mss,speed_ms,0,blend_radius_m)
    movel([0.080629, -1.231691, -2.664504, -0.816193, 1.570796, 1.651425],accel_mss,speed_ms,0,blend_radius_m)
    movel([0.080637, -1.231252, -2.664728, -0.816409, 1.570796, 1.651433],accel_mss,speed_ms,0,blend_radius_m)
    movel([0.080778, -1.230420, -2.665152, -0.816817, 1.570796, 1.651575],accel_mss,speed_ms,0,blend_radius_m)
    movel([0.080941, -1.229488, -2.665626, -0.817275, 1.570796, 1.651737],accel_mss,speed_ms,0,blend_radius_m)
    movel([0.080916, -1.229153, -2.665796, -0.817440, 1.570796, 1.651712],accel_mss,speed_ms,0,blend_radius_m)
    movel([0.080357, -1.229302, -2.665720, -0.817366, 1.570796, 1.651153],accel_mss,speed_ms,0,blend_radius_m)
    movel([0.079985, -1.229531, -2.665604, -0.817254, 1.570796, 1.650781],accel_mss,speed_ms,0,blend_radius_m)
    movel([0.079609, -1.229709, -2.665514, -0.817166, 1.570796, 1.650405],accel_mss,speed_ms,0,blend_radius_m)
    movel([0.079304, -1.229708, -2.665514, -0.817166, 1.570796, 1.650100],accel_mss,speed_ms,0,blend_radius_m)
    movel([0.079388, -1.229418, -2.665661, -0.817309, 1.570796, 1.650184],accel_mss,speed_ms,0,blend_radius_m)
    movel([0.079510, -1.228993, -2.665877, -0.817519, 1.570796, 1.650306],accel_mss,speed_ms,0,blend_radius_m)
    movel([0.079650, -1.228488, -2.666133, -0.817768, 1.570796, 1.650447],accel_mss,speed_ms,0,blend_radius_m)
    movel([0.079801, -1.227939, -2.666411, -0.818039, 1.570796, 1.650597],accel_mss,speed_ms,0,blend_radius_m)
    speed_ms = 0.003
    movel([0.079801, -1.213569, -2.659364, -0.839455, 1.570796, 1.650597],accel_mss,speed_ms,0,blend_radius_m)
    speed_ms = 1.000
    movel([0.079801, -1.186394, -2.644900, -0.881096, 1.570796, 1.650597],accel_mss,speed_ms,0,blend_radius_m)
    movel([0.085537, -1.198730, -2.638912, -0.874747, 1.570796, 1.656333],accel_mss,speed_ms,0,blend_radius_m)
    movel([0.085537, -1.225794, -2.653214, -0.833381, 1.570796, 1.656333],accel_mss,speed_ms,0,blend_radius_m)
    speed_ms = 0.003
    movel([0.085537, -1.236465, -2.658449, -0.817475, 1.570796, 1.656333],accel_mss,speed_ms,0,blend_radius_m)
    speed_ms = 0.007
    movel([0.086091, -1.236187, -2.658593, -0.817609, 1.570796, 1.656887],accel_mss,speed_ms,0,blend_radius_m)
    movel([0.086560, -1.236046, -2.658666, -0.817677, 1.570796, 1.657356],accel_mss,speed_ms,0,blend_radius_m)
    movel([0.086864, -1.236275, -2.658547, -0.817567, 1.570796, 1.657660],accel_mss,speed_ms,0,blend_radius_m)
    movel([0.086770, -1.236683, -2.658336, -0.817370, 1.570796, 1.657566],accel_mss,speed_ms,0,blend_radius_m)
    movel([0.086693, -1.236971, -2.658187, -0.817231, 1.570796, 1.657490],accel_mss,speed_ms,0,blend_radius_m)
    movel([0.086615, -1.237427, -2.657950, -0.817012, 1.570796, 1.657411],accel_mss,speed_ms,0,blend_radius_m)
    movel([0.086542, -1.237944, -2.657682, -0.816763, 1.570796, 1.657339],accel_mss,speed_ms,0,blend_radius_m)
    movel([0.086493, -1.238455, -2.657416, -0.816517, 1.570796, 1.657289],accel_mss,speed_ms,0,blend_radius_m)
    movel([0.086441, -1.238959, -2.657154, -0.816276, 1.570796, 1.657238],accel_mss,speed_ms,0,blend_radius_m)
    movel([0.086373, -1.239397, -2.656926, -0.816066, 1.570796, 1.657170],accel_mss,speed_ms,0,blend_radius_m)
    movel([0.086297, -1.239748, -2.656743, -0.815898, 1.570796, 1.657093],accel_mss,speed_ms,0,blend_radius_m)
    movel([0.085856, -1.240006, -2.656608, -0.815775, 1.570796, 1.656652],accel_mss,speed_ms,0,blend_radius_m)
    movel([0.085399, -1.239502, -2.656871, -0.816016, 1.570796, 1.656195],accel_mss,speed_ms,0,blend_radius_m)
    movel([0.085016, -1.238691, -2.657294, -0.816405, 1.570796, 1.655813],accel_mss,speed_ms,0,blend_radius_m)
    movel([0.084865, -1.237785, -2.657765, -0.816840, 1.570796, 1.655661],accel_mss,speed_ms,0,blend_radius_m)
    movel([0.084926, -1.237264, -2.658035, -0.817090, 1.570796, 1.655722],accel_mss,speed_ms,0,blend_radius_m)
    movel([0.085148, -1.236824, -2.658263, -0.817302, 1.570796, 1.655944],accel_mss,speed_ms,0,blend_radius_m)
    movel([0.085537, -1.236465, -2.658449, -0.817475, 1.570796, 1.656333],accel_mss,speed_ms,0,blend_radius_m)
    speed_ms = 0.003
    movel([0.085537, -1.240087, -2.660178, -0.812124, 1.570796, 1.656333],accel_mss,speed_ms,0,blend_radius_m)
    speed_ms = 0.007
    movel([0.086091, -1.239809, -2.660322, -0.812258, 1.570796, 1.656887],accel_mss,speed_ms,0,blend_radius_m)
    movel([0.086560, -1.239668, -2.660395, -0.812325, 1.570796, 1.657356],accel_mss,speed_ms,0,blend_radius_m)
    movel([0.086864, -1.239897, -2.660276, -0.812215, 1.570796, 1.657660],accel_mss,speed_ms,0,blend_radius_m)
    movel([0.086770, -1.240304, -2.660064, -0.812020, 1.570796, 1.657566],accel_mss,speed_ms,0,blend_radius_m)
    movel([0.086693, -1.240592, -2.659915, -0.811882, 1.570796, 1.657490],accel_mss,speed_ms,0,blend_radius_m)
    movel([0.086615, -1.241047, -2.659678, -0.811664, 1.570796, 1.657411],accel_mss,speed_ms,0,blend_radius_m)
    movel([0.086542, -1.241564, -2.659408, -0.811417, 1.570796, 1.657339],accel_mss,speed_ms,0,blend_radius_m)
    movel([0.086493, -1.242074, -2.659142, -0.811174, 1.570796, 1.657289],accel_mss,speed_ms,0,blend_radius_m)
    movel([0.086441, -1.242577, -2.658879, -0.810934, 1.570796, 1.657238],accel_mss,speed_ms,0,blend_radius_m)
    movel([0.086373, -1.243014, -2.658650, -0.810726, 1.570796, 1.657170],accel_mss,speed_ms,0,blend_radius_m)
    movel([0.086297, -1.243364, -2.658466, -0.810559, 1.570796, 1.657093],accel_mss,speed_ms,0,blend_radius_m)
    movel([0.085856, -1.243621, -2.658331, -0.810436, 1.570796, 1.656652],accel_mss,speed_ms,0,blend_radius_m)
    movel([0.085399, -1.243118, -2.658595, -0.810676, 1.570796, 1.656195],accel_mss,speed_ms,0,blend_radius_m)
    movel([0.085016, -1.242308, -2.659019, -0.811062, 1.570796, 1.655813],accel_mss,speed_ms,0,blend_radius_m)
    movel([0.084865, -1.241404, -2.659491, -0.811494, 1.570796, 1.655661],accel_mss,speed_ms,0,blend_radius_m)
    movel([0.084926, -1.240884, -2.659762, -0.811742, 1.570796, 1.655722],accel_mss,speed_ms,0,blend_radius_m)
    movel([0.085148, -1.240445, -2.659991, -0.811953, 1.570796, 1.655944],accel_mss,speed_ms,0,blend_radius_m)
    movel([0.085537, -1.240087, -2.660178, -0.812124, 1.570796, 1.656333],accel_mss,speed_ms,0,blend_radius_m)
    speed_ms = 0.003
    movel([0.085537, -1.225794, -2.653214, -0.833381, 1.570796, 1.656333],accel_mss,speed_ms,0,blend_radius_m)
    speed_ms = 1.000
    movel([0.085537, -1.198730, -2.638912, -0.874747, 1.570796, 1.656333],accel_mss,speed_ms,0,blend_radius_m)
    movel([0.087604, -1.198400, -2.639074, -0.874915, 1.570796, 1.658400],accel_mss,speed_ms,0,blend_radius_m)
    movel([0.087604, -1.225467, -2.653381, -0.833542, 1.570796, 1.658400],accel_mss,speed_ms,0,blend_radius_m)
    speed_ms = 0.003
    movel([0.087604, -1.236139, -2.658617, -0.817632, 1.570796, 1.658400],accel_mss,speed_ms,0,blend_radius_m)
    speed_ms = 0.007
    movel([0.087906, -1.235427, -2.658985, -0.817976, 1.570796, 1.658702],accel_mss,speed_ms,0,blend_radius_m)
    movel([0.088245, -1.234804, -2.659307, -0.818278, 1.570796, 1.659041],accel_mss,speed_ms,0,blend_radius_m)
    movel([0.088569, -1.234333, -2.659550, -0.818506, 1.570796, 1.659365],accel_mss,speed_ms,0,blend_radius_m)
    movel([0.088941, -1.234192, -2.659622, -0.818575, 1.570796, 1.659738],accel_mss,speed_ms,0,blend_radius_m)
    movel([0.088954, -1.234644, -2.659390, -0.818355, 1.570796, 1.659750],accel_mss,speed_ms,0,blend_radius_m)
    movel([0.088902, -1.235483, -2.658957, -0.817949, 1.570796, 1.659699],accel_mss,speed_ms,0,blend_radius_m)
    movel([0.088726, -1.237324, -2.658004, -0.817061, 1.570796, 1.659522],accel_mss,speed_ms,0,blend_radius_m)
    movel([0.088565, -1.238862, -2.657205, -0.816322, 1.570796, 1.659362],accel_mss,speed_ms,0,blend_radius_m)
    movel([0.088438, -1.239862, -2.656684, -0.815843, 1.570796, 1.659234],accel_mss,speed_ms,0,blend_radius_m)
    movel([0.088322, -1.240575, -2.656311, -0.815503, 1.570796, 1.659118],accel_mss,speed_ms,0,blend_radius_m)
    movel([0.087986, -1.240806, -2.656191, -0.815392, 1.570796, 1.658783],accel_mss,speed_ms,0,blend_radius_m)
    movel([0.087703, -1.240616, -2.656290, -0.815483, 1.570796, 1.658499],accel_mss,speed_ms,0,blend_radius_m)
    movel([0.087437, -1.240251, -2.656481, -0.815657, 1.570796, 1.658233],accel_mss,speed_ms,0,blend_radius_m)
    movel([0.087256, -1.239762, -2.656736, -0.815891, 1.570796, 1.658053],accel_mss,speed_ms,0,blend_radius_m)
    movel([0.087156, -1.239010, -2.657127, -0.816251, 1.570796, 1.657952],accel_mss,speed_ms,0,blend_radius_m)
    movel([0.087194, -1.238032, -2.657636, -0.816721, 1.570796, 1.657990],accel_mss,speed_ms,0,blend_radius_m)
    movel([0.087347, -1.237011, -2.658166, -0.817212, 1.570796, 1.658144],accel_mss,speed_ms,0,blend_radius_m)
    movel([0.087604, -1.236139, -2.658617, -0.817632, 1.570796, 1.658400],accel_mss,speed_ms,0,blend_radius_m)
    speed_ms = 0.003
    movel([0.087604, -1.239762, -2.660347, -0.812281, 1.570796, 1.658400],accel_mss,speed_ms,0,blend_radius_m)
    speed_ms = 0.007
    movel([0.087906, -1.239051, -2.660716, -0.812622, 1.570796, 1.658702],accel_mss,speed_ms,0,blend_radius_m)
    movel([0.088245, -1.238429, -2.661039, -0.812922, 1.570796, 1.659041],accel_mss,speed_ms,0,blend_radius_m)
    movel([0.088569, -1.237958, -2.661283, -0.813148, 1.570796, 1.659365],accel_mss,speed_ms,0,blend_radius_m)
    movel([0.088941, -1.237817, -2.661355, -0.813216, 1.570796, 1.659738],accel_mss,speed_ms,0,blend_radius_m)
    movel([0.088954, -1.238269, -2.661122, -0.812999, 1.570796, 1.659750],accel_mss,speed_ms,0,blend_radius_m)
    movel([0.088902, -1.239106, -2.660687, -0.812595, 1.570796, 1.659699],accel_mss,speed_ms,0,blend_radius_m)
    movel([0.088726, -1.240944, -2.659731, -0.811714, 1.570796, 1.659522],accel_mss,speed_ms,0,blend_radius_m)
    movel([0.088565, -1.242479, -2.658930, -0.810980, 1.570796, 1.659362],accel_mss,speed_ms,0,blend_radius_m)
    movel([0.088438, -1.243478, -2.658407, -0.810505, 1.570796, 1.659234],accel_mss,speed_ms,0,blend_radius_m)
    movel([0.088322, -1.244190, -2.658033, -0.810166, 1.570796, 1.659118],accel_mss,speed_ms,0,blend_radius_m)
    movel([0.087986, -1.244420, -2.657912, -0.810057, 1.570796, 1.658783],accel_mss,speed_ms,0,blend_radius_m)
    movel([0.087703, -1.244230, -2.658012, -0.810147, 1.570796, 1.658499],accel_mss,speed_ms,0,blend_radius_m)
    movel([0.087437, -1.243866, -2.658203, -0.810320, 1.570796, 1.658233],accel_mss,speed_ms,0,blend_radius_m)
    movel([0.087256, -1.243378, -2.658459, -0.810552, 1.570796, 1.658053],accel_mss,speed_ms,0,blend_radius_m)
    movel([0.087156, -1.242628, -2.658852, -0.810909, 1.570796, 1.657952],accel_mss,speed_ms,0,blend_radius_m)
    movel([0.087194, -1.241651, -2.659363, -0.811376, 1.570796, 1.657990],accel_mss,speed_ms,0,blend_radius_m)
    movel([0.087347, -1.240632, -2.659894, -0.811863, 1.570796, 1.658144],accel_mss,speed_ms,0,blend_radius_m)
    movel([0.087604, -1.239762, -2.660347, -0.812281, 1.570796, 1.658400],accel_mss,speed_ms,0,blend_radius_m)
    speed_ms = 0.003
    movel([0.087604, -1.225467, -2.653381, -0.833542, 1.570796, 1.658400],accel_mss,speed_ms,0,blend_radius_m)
    speed_ms = 1.000
    movel([0.087604, -1.198400, -2.639074, -0.874915, 1.570796, 1.658400],accel_mss,speed_ms,0,blend_radius_m)
    movel([0.099050, -1.197856, -2.639341, -0.875191, 1.570796, 1.669847],accel_mss,speed_ms,0,blend_radius_m)
    movel([0.099050, -1.224928, -2.653655, -0.833806, 1.570796, 1.669847],accel_mss,speed_ms,0,blend_radius_m)
    speed_ms = 0.003
    movel([0.099050, -1.235604, -2.658894, -0.817891, 1.570796, 1.669847],accel_mss,speed_ms,0,blend_radius_m)
    speed_ms = 0.007
    movel([0.099408, -1.235304, -2.659049, -0.818036, 1.570796, 1.670205],accel_mss,speed_ms,0,blend_radius_m)
    movel([0.099751, -1.235327, -2.659037, -0.818025, 1.570796, 1.670547],accel_mss,speed_ms,0,blend_radius_m)
    movel([0.099887, -1.235536, -2.658929, -0.817924, 1.570796, 1.670683],accel_mss,speed_ms,0,blend_radius_m)
    movel([0.099641, -1.235906, -2.658738, -0.817745, 1.570796, 1.670437],accel_mss,speed_ms,0,blend_radius_m)
    movel([0.099319, -1.236141, -2.658617, -0.817632, 1.570796, 1.670115],accel_mss,speed_ms,0,blend_radius_m)
    movel([0.099022, -1.236150, -2.658612, -0.817627, 1.570796, 1.669818],accel_mss,speed_ms,0,blend_radius_m)
    movel([0.098912, -1.235929, -2.658726, -0.817734, 1.570796, 1.669708],accel_mss,speed_ms,0,blend_radius_m)
    movel([0.099050, -1.235604, -2.658894, -0.817891, 1.570796, 1.669847],accel_mss,speed_ms,0,blend_radius_m)
    speed_ms = 0.003
    movel([0.099050, -1.239227, -2.660625, -0.812538, 1.570796, 1.669847],accel_mss,speed_ms,0,blend_radius_m)
    speed_ms = 0.007
    movel([0.099408, -1.238928, -2.660780, -0.812681, 1.570796, 1.670205],accel_mss,speed_ms,0,blend_radius_m)
    movel([0.099751, -1.238951, -2.660768, -0.812670, 1.570796, 1.670547],accel_mss,speed_ms,0,blend_radius_m)
    movel([0.099887, -1.239159, -2.660660, -0.812570, 1.570796, 1.670683],accel_mss,speed_ms,0,blend_radius_m)
    movel([0.099641, -1.239529, -2.660468, -0.812392, 1.570796, 1.670437],accel_mss,speed_ms,0,blend_radius_m)
    movel([0.099319, -1.239763, -2.660346, -0.812280, 1.570796, 1.670115],accel_mss,speed_ms,0,blend_radius_m)
    movel([0.099022, -1.239772, -2.660341, -0.812275, 1.570796, 1.669818],accel_mss,speed_ms,0,blend_radius_m)
    movel([0.098912, -1.239552, -2.660456, -0.812381, 1.570796, 1.669708],accel_mss,speed_ms,0,blend_radius_m)
    movel([0.099050, -1.239227, -2.660625, -0.812538, 1.570796, 1.669847],accel_mss,speed_ms,0,blend_radius_m)
    speed_ms = 0.003
    movel([0.099050, -1.224928, -2.653655, -0.833806, 1.570796, 1.669847],accel_mss,speed_ms,0,blend_radius_m)
    speed_ms = 1.000
    movel([0.099050, -1.197856, -2.639341, -0.875191, 1.570796, 1.669847],accel_mss,speed_ms,0,blend_radius_m)
    movel([0.101409, -1.195286, -2.640600, -0.876503, 1.570796, 1.672205],accel_mss,speed_ms,0,blend_radius_m)
    movel([0.101409, -1.222382, -2.654947, -0.835059, 1.570796, 1.672205],accel_mss,speed_ms,0,blend_radius_m)
    speed_ms = 0.003
    movel([0.101409, -1.233070, -2.660200, -0.819120, 1.570796, 1.672205],accel_mss,speed_ms,0,blend_radius_m)
    speed_ms = 0.007
    movel([0.102317, -1.234124, -2.659657, -0.818608, 1.570796, 1.673113],accel_mss,speed_ms,0,blend_radius_m)
    movel([0.102472, -1.234924, -2.659245, -0.818220, 1.570796, 1.673268],accel_mss,speed_ms,0,blend_radius_m)
    movel([0.102400, -1.235927, -2.658727, -0.817735, 1.570796, 1.673197],accel_mss,speed_ms,0,blend_radius_m)
    movel([0.102133, -1.236981, -2.658181, -0.817226, 1.570796, 1.672929],accel_mss,speed_ms,0,blend_radius_m)
    movel([0.101697, -1.237925, -2.657692, -0.816772, 1.570796, 1.672493],accel_mss,speed_ms,0,blend_radius_m)
    movel([0.100068, -1.239955, -2.656635, -0.815799, 1.570796, 1.670864],accel_mss,speed_ms,0,blend_radius_m)
    movel([0.097976, -1.241450, -2.655854, -0.815085, 1.570796, 1.668772],accel_mss,speed_ms,0,blend_radius_m)
    movel([0.095827, -1.242120, -2.655503, -0.814766, 1.570796, 1.666623],accel_mss,speed_ms,0,blend_radius_m)
    movel([0.094036, -1.241842, -2.655648, -0.814899, 1.570796, 1.664832],accel_mss,speed_ms,0,blend_radius_m)
    movel([0.093156, -1.241077, -2.656049, -0.815263, 1.570796, 1.663953],accel_mss,speed_ms,0,blend_radius_m)
    movel([0.092741, -1.239931, -2.656648, -0.815811, 1.570796, 1.663537],accel_mss,speed_ms,0,blend_radius_m)
    movel([0.092831, -1.238531, -2.657377, -0.816481, 1.570796, 1.663628],accel_mss,speed_ms,0,blend_radius_m)
    movel([0.093422, -1.237038, -2.658152, -0.817199, 1.570796, 1.664218],accel_mss,speed_ms,0,blend_radius_m)
    movel([0.093877, -1.236345, -2.658511, -0.817533, 1.570796, 1.664673],accel_mss,speed_ms,0,blend_radius_m)
    movel([0.094527, -1.235561, -2.658916, -0.817912, 1.570796, 1.665323],accel_mss,speed_ms,0,blend_radius_m)
    movel([0.095260, -1.234808, -2.659305, -0.818276, 1.570796, 1.666057],accel_mss,speed_ms,0,blend_radius_m)
    movel([0.095976, -1.234201, -2.659618, -0.818570, 1.570796, 1.666773],accel_mss,speed_ms,0,blend_radius_m)
    movel([0.097903, -1.233111, -2.660179, -0.819100, 1.570796, 1.668700],accel_mss,speed_ms,0,blend_radius_m)
    movel([0.099837, -1.232714, -2.660382, -0.819293, 1.570796, 1.670633],accel_mss,speed_ms,0,blend_radius_m)
    movel([0.101409, -1.233070, -2.660200, -0.819120, 1.570796, 1.672205],accel_mss,speed_ms,0,blend_radius_m)
    speed_ms = 0.003
    movel([0.101409, -1.236697, -2.661934, -0.813757, 1.570796, 1.672205],accel_mss,speed_ms,0,blend_radius_m)
    speed_ms = 0.007
    movel([0.102317, -1.237750, -2.661390, -0.813249, 1.570796, 1.673113],accel_mss,speed_ms,0,blend_radius_m)
    movel([0.102472, -1.238548, -2.660977, -0.812864, 1.570796, 1.673268],accel_mss,speed_ms,0,blend_radius_m)
    movel([0.102400, -1.239550, -2.660457, -0.812382, 1.570796, 1.673197],accel_mss,speed_ms,0,blend_radius_m)
    movel([0.102133, -1.240602, -2.659909, -0.811877, 1.570796, 1.672929],accel_mss,speed_ms,0,blend_radius_m)
    movel([0.101697, -1.241544, -2.659418, -0.811427, 1.570796, 1.672493],accel_mss,speed_ms,0,blend_radius_m)
    movel([0.100068, -1.243571, -2.658358, -0.810460, 1.570796, 1.670864],accel_mss,speed_ms,0,blend_radius_m)
    movel([0.097976, -1.245063, -2.657574, -0.809752, 1.570796, 1.668772],accel_mss,speed_ms,0,blend_radius_m)
    movel([0.095827, -1.245732, -2.657222, -0.809435, 1.570796, 1.666623],accel_mss,speed_ms,0,blend_radius_m)
    movel([0.094036, -1.245454, -2.657368, -0.809567, 1.570796, 1.664832],accel_mss,speed_ms,0,blend_radius_m)
    movel([0.093156, -1.244691, -2.657770, -0.809928, 1.570796, 1.663953],accel_mss,speed_ms,0,blend_radius_m)
    movel([0.092741, -1.243546, -2.658371, -0.810472, 1.570796, 1.663537],accel_mss,speed_ms,0,blend_radius_m)
    movel([0.092831, -1.242149, -2.659102, -0.811138, 1.570796, 1.663628],accel_mss,speed_ms,0,blend_radius_m)
    movel([0.093422, -1.240659, -2.659880, -0.811850, 1.570796, 1.664218],accel_mss,speed_ms,0,blend_radius_m)
    movel([0.093877, -1.239967, -2.660240, -0.812182, 1.570796, 1.664673],accel_mss,speed_ms,0,blend_radius_m)
    movel([0.094527, -1.239184, -2.660647, -0.812558, 1.570796, 1.665323],accel_mss,speed_ms,0,blend_radius_m)
    movel([0.095260, -1.238433, -2.661037, -0.812920, 1.570796, 1.666057],accel_mss,speed_ms,0,blend_radius_m)
    movel([0.095976, -1.237826, -2.661351, -0.813212, 1.570796, 1.666773],accel_mss,speed_ms,0,blend_radius_m)
    movel([0.097903, -1.236738, -2.661913, -0.813738, 1.570796, 1.668700],accel_mss,speed_ms,0,blend_radius_m)
    movel([0.099837, -1.236342, -2.662118, -0.813929, 1.570796, 1.670633],accel_mss,speed_ms,0,blend_radius_m)
    movel([0.101409, -1.236697, -2.661934, -0.813757, 1.570796, 1.672205],accel_mss,speed_ms,0,blend_radius_m)
    speed_ms = 0.003
    movel([0.101409, -1.222382, -2.654947, -0.835059, 1.570796, 1.672205],accel_mss,speed_ms,0,blend_radius_m)
    speed_ms = 1.000
    movel([0.101409, -1.195286, -2.640600, -0.876503, 1.570796, 1.672205],accel_mss,speed_ms,0,blend_radius_m)
    movel([0.111071, -1.194203, -2.641128, -0.877058, 1.570796, 1.681867],accel_mss,speed_ms,0,blend_radius_m)
    movel([0.111071, -1.221309, -2.655490, -0.835590, 1.570796, 1.681867],accel_mss,speed_ms,0,blend_radius_m)
    speed_ms = 0.003
    movel([0.111071, -1.232002, -2.660748, -0.819640, 1.570796, 1.681867],accel_mss,speed_ms,0,blend_radius_m)
    speed_ms = 0.007
    movel([0.111227, -1.231656, -2.660925, -0.819808, 1.570796, 1.682024],accel_mss,speed_ms,0,blend_radius_m)
    movel([0.111558, -1.231401, -2.661055, -0.819933, 1.570796, 1.682354],accel_mss,speed_ms,0,blend_radius_m)
    movel([0.111877, -1.231380, -2.661066, -0.819943, 1.570796, 1.682673],accel_mss,speed_ms,0,blend_radius_m)
    movel([0.111993, -1.231681, -2.660912, -0.819796, 1.570796, 1.682790],accel_mss,speed_ms,0,blend_radius_m)
    movel([0.111655, -1.232138, -2.660678, -0.819573, 1.570796, 1.682452],accel_mss,speed_ms,0,blend_radius_m)
    movel([0.111288, -1.232299, -2.660595, -0.819495, 1.570796, 1.682084],accel_mss,speed_ms,0,blend_radius_m)
    movel([0.111071, -1.232002, -2.660748, -0.819640, 1.570796, 1.681867],accel_mss,speed_ms,0,blend_radius_m)
    speed_ms = 0.003
    movel([0.111071, -1.235631, -2.662484, -0.814274, 1.570796, 1.681867],accel_mss,speed_ms,0,blend_radius_m)
    speed_ms = 0.007
    movel([0.111227, -1.235286, -2.662662, -0.814441, 1.570796, 1.682024],accel_mss,speed_ms,0,blend_radius_m)
    movel([0.111558, -1.235032, -2.662793, -0.814565, 1.570796, 1.682354],accel_mss,speed_ms,0,blend_radius_m)
    movel([0.111877, -1.235010, -2.662804, -0.814575, 1.570796, 1.682673],accel_mss,speed_ms,0,blend_radius_m)
    movel([0.111993, -1.235311, -2.662649, -0.814429, 1.570796, 1.682790],accel_mss,speed_ms,0,blend_radius_m)
    movel([0.111655, -1.235767, -2.662414, -0.814208, 1.570796, 1.682452],accel_mss,speed_ms,0,blend_radius_m)
    movel([0.111288, -1.235928, -2.662331, -0.814130, 1.570796, 1.682084],accel_mss,speed_ms,0,blend_radius_m)
    movel([0.111071, -1.235631, -2.662484, -0.814274, 1.570796, 1.681867],accel_mss,speed_ms,0,blend_radius_m)
    speed_ms = 0.003
    movel([0.111071, -1.221309, -2.655490, -0.835590, 1.570796, 1.681867],accel_mss,speed_ms,0,blend_radius_m)
    speed_ms = 1.000
    movel([0.111071, -1.194203, -2.641128, -0.877058, 1.570796, 1.681867],accel_mss,speed_ms,0,blend_radius_m)
    movel([0.109412, -1.193393, -2.641522, -0.877474, 1.570796, 1.680209],accel_mss,speed_ms,0,blend_radius_m)
    movel([0.109412, -1.220507, -2.655895, -0.835988, 1.570796, 1.680209],accel_mss,speed_ms,0,blend_radius_m)
    speed_ms = 0.003
    movel([0.109412, -1.231203, -2.661157, -0.820030, 1.570796, 1.680209],accel_mss,speed_ms,0,blend_radius_m)
    speed_ms = 0.007
    movel([0.110087, -1.230365, -2.661585, -0.820439, 1.570796, 1.680884],accel_mss,speed_ms,0,blend_radius_m)
    movel([0.110838, -1.229594, -2.661978, -0.820817, 1.570796, 1.681634],accel_mss,speed_ms,0,blend_radius_m)
    movel([0.111575, -1.228983, -2.662289, -0.821117, 1.570796, 1.682372],accel_mss,speed_ms,0,blend_radius_m)
    movel([0.113674, -1.227893, -2.662843, -0.821653, 1.570796, 1.684470],accel_mss,speed_ms,0,blend_radius_m)
    movel([0.115711, -1.227621, -2.662981, -0.821787, 1.570796, 1.686507],accel_mss,speed_ms,0,blend_radius_m)
    movel([0.117256, -1.228220, -2.662677, -0.821492, 1.570796, 1.688052],accel_mss,speed_ms,0,blend_radius_m)
    movel([0.117989, -1.229566, -2.661992, -0.820830, 1.570796, 1.688785],accel_mss,speed_ms,0,blend_radius_m)
    movel([0.117965, -1.230677, -2.661426, -0.820287, 1.570796, 1.688761],accel_mss,speed_ms,0,blend_radius_m)
    movel([0.117577, -1.231979, -2.660759, -0.819651, 1.570796, 1.688373],accel_mss,speed_ms,0,blend_radius_m)
    movel([0.116887, -1.233303, -2.660080, -0.819006, 1.570796, 1.687683],accel_mss,speed_ms,0,blend_radius_m)
    movel([0.115976, -1.234480, -2.659474, -0.818435, 1.570796, 1.686772],accel_mss,speed_ms,0,blend_radius_m)
    movel([0.115156, -1.235287, -2.659058, -0.818044, 1.570796, 1.685952],accel_mss,speed_ms,0,blend_radius_m)
    movel([0.114390, -1.235879, -2.658752, -0.817758, 1.570796, 1.685186],accel_mss,speed_ms,0,blend_radius_m)
    movel([0.113558, -1.236344, -2.658512, -0.817534, 1.570796, 1.684355],accel_mss,speed_ms,0,blend_radius_m)
    movel([0.112538, -1.236756, -2.658298, -0.817335, 1.570796, 1.683335],accel_mss,speed_ms,0,blend_radius_m)
    movel([0.111513, -1.237055, -2.658143, -0.817191, 1.570796, 1.682309],accel_mss,speed_ms,0,blend_radius_m)
    movel([0.110720, -1.237150, -2.658094, -0.817145, 1.570796, 1.681516],accel_mss,speed_ms,0,blend_radius_m)
    movel([0.110024, -1.237046, -2.658148, -0.817195, 1.570796, 1.680820],accel_mss,speed_ms,0,blend_radius_m)
    movel([0.109302, -1.236738, -2.658307, -0.817344, 1.570796, 1.680098],accel_mss,speed_ms,0,blend_radius_m)
    movel([0.108717, -1.236294, -2.658537, -0.817558, 1.570796, 1.679513],accel_mss,speed_ms,0,blend_radius_m)
    movel([0.108365, -1.235748, -2.658820, -0.817822, 1.570796, 1.679162],accel_mss,speed_ms,0,blend_radius_m)
    movel([0.108218, -1.235030, -2.659190, -0.818169, 1.570796, 1.679014],accel_mss,speed_ms,0,blend_radius_m)
    movel([0.108256, -1.234068, -2.659686, -0.818635, 1.570796, 1.679053],accel_mss,speed_ms,0,blend_radius_m)
    movel([0.108349, -1.233414, -2.660023, -0.818952, 1.570796, 1.679145],accel_mss,speed_ms,0,blend_radius_m)
    movel([0.108457, -1.232964, -2.660254, -0.819171, 1.570796, 1.679253],accel_mss,speed_ms,0,blend_radius_m)
    movel([0.108621, -1.232542, -2.660470, -0.819376, 1.570796, 1.679418],accel_mss,speed_ms,0,blend_radius_m)
    movel([0.108896, -1.232009, -2.660744, -0.819636, 1.570796, 1.679692],accel_mss,speed_ms,0,blend_radius_m)
    movel([0.109412, -1.231203, -2.661157, -0.820030, 1.570796, 1.680209],accel_mss,speed_ms,0,blend_radius_m)
    speed_ms = 0.003
    movel([0.109412, -1.234833, -2.662895, -0.814661, 1.570796, 1.680209],accel_mss,speed_ms,0,blend_radius_m)
    speed_ms = 0.007
    movel([0.110087, -1.233997, -2.663324, -0.815068, 1.570796, 1.680884],accel_mss,speed_ms,0,blend_radius_m)
    movel([0.110838, -1.233227, -2.663719, -0.815443, 1.570796, 1.681634],accel_mss,speed_ms,0,blend_radius_m)
    movel([0.111575, -1.232617, -2.664031, -0.815741, 1.570796, 1.682372],accel_mss,speed_ms,0,blend_radius_m)
    movel([0.113674, -1.231529, -2.664587, -0.816273, 1.570796, 1.684470],accel_mss,speed_ms,0,blend_radius_m)
